  STRUCT
   S700 : STRUCT
    M_AUTO_SEL : BOOL ;
    M_MANUAL_SEL : BOOL ;
    M_READY_PB : BOOL ;
    M_AUTO_RUN_PB : BOOL ;
    M_WORK_COMP_SET_PB : BOOL ;
    M_WORK_COMP_RST_PB : BOOL ;
    M_HOME_POS_PB : BOOL ;
    SPARE8 : BOOL ;
    TL_PIN_SEL : BOOL ;
    LM_PIN_SEL : BOOL ;
    TL_LATCH_SEL : BOOL ;
    LM_LATCH_SEL : BOOL ;
    SPARE13 : BOOL ;
    SPARE14 : BOOL ;
    SPARE15 : BOOL ;
    SPARE16 : BOOL ;
    SPARE17 : BOOL ;
    SPARE18 : BOOL ;
    SPARE19 : BOOL ;
    SPARE20 : BOOL ;
    SPARE21 : BOOL ;
    SPARE22 : BOOL ;
    SPARE23 : BOOL ;
    SPARE24 : BOOL ;
    SPARE25 : BOOL ;
    SPARE26 : BOOL ;
    SPARE27 : BOOL ;
    SPARE28 : BOOL ;
    SPARE29 : BOOL ;
    SPARE30 : BOOL ;
    M_ADV_PB : BOOL ;
    M_RET_PB : BOOL ;
    SPARE34 : BOOL ;
    SPARE35 : BOOL ;
    SPARE36 : BOOL ;
    SPARE37 : BOOL ;
    M_RBT_WORK_COMP_SET_PB : BOOL ;
    M_RBT_WORK_COMP_RST_PB : BOOL ;
    SPARE40 : BOOL ;
    SPARE41 : BOOL ;
    SPARE42 : BOOL ;
    SPARE43 : BOOL ;
    SPARE44 : BOOL ;
    SPARE45 : BOOL ;
    SPARE46 : BOOL ;
    SPARE47 : BOOL ;
    SPARE48 : BOOL ;
    SPARE49 : BOOL ;
    SPARE50 : BOOL ;
    SPARE51 : BOOL ;
    SPARE52 : BOOL ;
    SPARE53 : BOOL ;
    SPARE54 : BOOL ;
    SPARE55 : BOOL ;
    SPARE56 : BOOL ;
    SPARE57 : BOOL ;
    SPARE58 : BOOL ;
    SPARE59 : BOOL ;
    SPARE60 : BOOL ;
    SPARE61 : BOOL ;
    SPARE62 : BOOL ;
    SPARE63 : BOOL ;
    SPARE64 : BOOL ;
    SPARE65 : BOOL ;
    SPARE66 : BOOL ;
    SPARE67 : BOOL ;
    SPARE68 : BOOL ;
    SPARE69 : BOOL ;
    SPARE70 : BOOL ;
    SPARE71 : BOOL ;
    SPARE72 : BOOL ;
    SPARE73 : BOOL ;
    SPARE74 : BOOL ;
    SPARE75 : BOOL ;
    SPARE76 : BOOL ;
    SPARE77 : BOOL ;
    SPARE78 : BOOL ;
    SPARE79 : BOOL ;
    SPARE80 : BOOL ;
    SPARE81 : BOOL ;
    SPARE82 : BOOL ;
    SPARE83 : BOOL ;
    SPARE84 : BOOL ;
    SPARE85 : BOOL ;
    SPARE86 : BOOL ;
    SPARE87 : BOOL ;
    SPARE88 : BOOL ;
    SPARE89 : BOOL ;
    SPARE90 : BOOL ;
    SPARE91 : BOOL ;
    SPARE92 : BOOL ;
    SPARE93 : BOOL ;
    SPARE94 : BOOL ;
    SPARE95 : BOOL ;
    SPARE96 : BOOL ;
    SPARE97 : BOOL ;
    SPARE98 : BOOL ;
    SPARE99 : BOOL ;
    SPARE100 : BOOL ;
    SPARE101 : BOOL ;
    SPARE102 : BOOL ;
    SPARE103 : BOOL ;
    SPARE104 : BOOL ;
    SPARE105 : BOOL ;
    SPARE106 : BOOL ;
    SPARE107 : BOOL ;
    SPARE108 : BOOL ;
    SPARE109 : BOOL ;
    SPARE110 : BOOL ;
    SPARE111 : BOOL ;
    SPARE112 : BOOL ;
    SPARE113 : BOOL ;
    SPARE114 : BOOL ;
    SPARE115 : BOOL ;
    SPARE116 : BOOL ;
    SPARE117 : BOOL ;
    SPARE118 : BOOL ;
    SPARE119 : BOOL ;
    SPARE120 : BOOL ;
    SPARE121 : BOOL ;
    SPARE122 : BOOL ;
    SPARE123 : BOOL ;
    SPARE124 : BOOL ;
    SPARE125 : BOOL ;
    SPARE126 : BOOL ;
    SPARE127 : BOOL ;
    SPARE128 : BOOL ;
    SPARE129 : BOOL ;
    SPARE130 : BOOL ;
    SPARE131 : BOOL ;
    SPARE132 : BOOL ;
    SPARE133 : BOOL ;
    SPARE134 : BOOL ;
    SPARE135 : BOOL ;
    SPARE136 : BOOL ;
    SPARE137 : BOOL ;
    SPARE138 : BOOL ;
    SPARE139 : BOOL ;
    SPARE140 : BOOL ;
    SPARE141 : BOOL ;
    SPARE142 : BOOL ;
    SPARE143 : BOOL ;
    SPARE144 : BOOL ;
    SPARE145 : BOOL ;
    SPARE146 : BOOL ;
    SPARE147 : BOOL ;
    SPARE148 : BOOL ;
    SPARE149 : BOOL ;
    SPARE150 : BOOL ;
    SPARE151 : BOOL ;
    SPARE152 : BOOL ;
    SPARE153 : BOOL ;
    SPARE154 : BOOL ;
    SPARE155 : BOOL ;
    SPARE156 : BOOL ;
    SPARE157 : BOOL ;
    SPARE158 : BOOL ;
    SPARE159 : BOOL ;
    SPARE160 : BOOL ;
    SPARE161 : BOOL ;
    TL_PIN_UP_LAMP : WORD ;
    TL_PIN_DOWN_LAMP : WORD ;
    LM_PIN_UP_LAMP : WORD ;
    LM_PIN_DOWN_LAMP : WORD ;
    TL_LATCH_ADV_LAMP : WORD ;
    TL_LATCH_RET_LAMP : WORD ;
    LM_LATCH_ADV_LAMP : WORD ;
    LM_LATCH_RET_LAMP : WORD ;
    SP_WORD19 : WORD ;
    SP_WORD20 : WORD ;
    SP_WORD21 : WORD ;
    SP_WORD22 : WORD ;
    SP_WORD23 : WORD ;
    SP_WORD24 : WORD ;
    SP_WORD25 : WORD ;
    SP_WORD26 : WORD ;
    SP_WORD27 : WORD ;
    SP_WORD28 : WORD ;
    SP_WORD29 : WORD ;
    SP_WORD30 : WORD ;
    SP_WORD31 : WORD ;
    SP_WORD32 : WORD ;
    SP_WORD33 : WORD ;
    SP_WORD34 : WORD ;
    SP_WORD36 : WORD ;
    SP_WORD37 : WORD ;
    SP_WORD38 : WORD ;
    SP_WORD39 : WORD ;
    SP_WORD40 : WORD ;
    SP_WORD41 : WORD ;
    SP_WORD42 : WORD ;
    SP_WORD43 : WORD ;
    SP_WORD44 : WORD ;
    SP_WORD45 : WORD ;
    SP_WORD46 : WORD ;
    SP_WORD47 : WORD ;
    SP_WORD48 : WORD ;
    SP_WORD49 : WORD ;
    SP_WORD50 : WORD ;
    SP_WORD51 : WORD ;
    SP_WORD52 : WORD ;
    SP_WORD53 : WORD ;
    SP_WORD54 : WORD ;
    SP_WORD55 : WORD ;
    SP_WORD56 : WORD ;
    SP_WORD57 : WORD ;
    SP_WORD58 : WORD ;
    SP_WORD59 : WORD ;
    SP_WORD60 : WORD ;
    SP_WORD61 : WORD ;
    SP_WORD62 : WORD ;
    SP_WORD63 : WORD ;
    SP_WORD64 : WORD ;
    SP_WORD65 : WORD ;
    SP_WORD66 : WORD ;
    SP_WORD67 : WORD ;
    SP_WORD68 : WORD ;
    SP_WORD69 : WORD ;
    SP_WORD70 : WORD ;
    SP_WORD71 : WORD ;
    SP_WORD72 : WORD ;
    SP_WORD73 : WORD ;
    SP_WORD74 : WORD ;
    SP_WORD75 : WORD ;
    SP_WORD76 : WORD ;
    SP_WORD77 : WORD ;
    SP_WORD78 : WORD ;
    SP_WORD79 : WORD ;
    SP_WORD80 : WORD ;
    SP_WORD81 : WORD ;
    SP_WORD82 : WORD ;
    SP_WORD83 : WORD ;
    SP_WORD84 : WORD ;
    SP_WORD85 : WORD ;
    SP_WORD86 : WORD ;
    SP_WORD87 : WORD ;
    SP_WORD88 : WORD ;
    SP_WORD89 : WORD ;
    SP_WORD90 : WORD ;
    SP_WORD91 : WORD ;
    SP_WORD92 : WORD ;
    SP_WORD93 : WORD ;
    SP_WORD94 : WORD ;
    SP_WORD95 : WORD ;
    SP_WORD96 : WORD ;
    SP_WORD97 : WORD ;
    SP_WORD98 : WORD ;
    SP_WORD99 : WORD ;
    SP_WORD100 : WORD ;
    SP_WORD101 : WORD ;
   END_STRUCT ;
   S701 : STRUCT
    M_AUTO_SEL : BOOL ;
    M_MANUAL_SEL : BOOL ;
    M_READY_PB : BOOL ;
    M_AUTO_RUN_PB : BOOL ;
    M_WORK_COMP_SET_PB : BOOL ;
    M_WORK_COMP_RST_PB : BOOL ;
    M_HOME_POS_PB : BOOL ;
    M_TIP_DRESS_PB : BOOL ;
    INDEX_RET_LOCK_SEL : BOOL ;
    INDEX_ADV_RET_SEL : BOOL ;
    INDEX_ADV_LOCK_SEL : BOOL ;
    SPARE12 : BOOL ;
    SPARE13 : BOOL ;
    SPARE14 : BOOL ;
    SPARE15 : BOOL ;
    SPARE16 : BOOL ;
    SPARE17 : BOOL ;
    SPARE18 : BOOL ;
    SPARE19 : BOOL ;
    SPARE20 : BOOL ;
    SPARE21 : BOOL ;
    SPARE22 : BOOL ;
    SPARE23 : BOOL ;
    SPARE24 : BOOL ;
    SPARE25 : BOOL ;
    SPARE26 : BOOL ;
    SPARE27 : BOOL ;
    SPARE28 : BOOL ;
    SPARE29 : BOOL ;
    SPARE30 : BOOL ;
    M_ADV_PB : BOOL ;
    M_RET_PB : BOOL ;
    LM_INDEX_PIN1_SEL : BOOL ;
    LM_INDEX_PIN2_SEL : BOOL ;
    LM_INDEX_PIN3_SEL : BOOL ;
    LM_INDEX_1_CLAMP1_SEL : BOOL ;
    LM_INDEX_1_CLAMP2_SEL : BOOL ;
    LM_INDEX_1_CLAMP3_SEL : BOOL ;
    LM_INDEX_1_CLAMP4_SEL : BOOL ;
    LM_INDEX_2_CLAMP1_SEL : BOOL ;
    LM_INDEX_2_CLAMP2_SEL : BOOL ;
    LM_INDEX_2_CLAMP3_SEL : BOOL ;
    LM_INDEX_2_CLAMP4_SEL : BOOL ;
    LM_INDEX_2_CLAMP5_SEL : BOOL ;
    LM_INDEX_FDR_SHIFT_SEL : BOOL ;
    LM_INDEX_FDR_PIN_SEL : BOOL ;
    LM_INDEX_ADV_PB : BOOL ;
    LM_INDEX_RET_PB : BOOL ;
    TL_INDEX_PIN1_SEL : BOOL ;
    TL_INDEX_PIN2_SEL : BOOL ;
    TL_INDEX_LOCATE1_SEL : BOOL ;
    TL_INDEX_LOCATE2_SEL : BOOL ;
    TL_INDEX_LOCATE3_SEL : BOOL ;
    TL_INDEX_1_CLAMP1_SEL : BOOL ;
    TL_INDEX_1_CLAMP2_SEL : BOOL ;
    TL_INDEX_CLAMP2_SEL : BOOL ;
    TL_INDEX_CLAMP3_SEL : BOOL ;
    TL_INDEX_CLAMP4_SEL : BOOL ;
    TL_INDEX_FDR_SHIFT_SEL : BOOL ;
    SPARE61 : BOOL ;
    SPARE62 : BOOL ;
    SPARE63 : BOOL ;
    TL_INDEX_ADV_PB : BOOL ;
    TL_INDEX_RET_PB : BOOL ;
    SPARE66 : BOOL ;
    SPARE67 : BOOL ;
    SPARE68 : BOOL ;
    SPARE69 : BOOL ;
    SPARE70 : BOOL ;
    SPARE71 : BOOL ;
    SPARE72 : BOOL ;
    SPARE73 : BOOL ;
    SPARE74 : BOOL ;
    SPARE75 : BOOL ;
    SPARE76 : BOOL ;
    SPARE77 : BOOL ;
    SPARE78 : BOOL ;
    SPARE79 : BOOL ;
    SPARE80 : BOOL ;
    SPARE81 : BOOL ;
    SPARE82 : BOOL ;
    SPARE83 : BOOL ;
    SPARE84 : BOOL ;
    SPARE85 : BOOL ;
    SPARE86 : BOOL ;
    SPARE87 : BOOL ;
    SPARE88 : BOOL ;
    SPARE89 : BOOL ;
    SPARE90 : BOOL ;
    SPARE91 : BOOL ;
    SPARE92 : BOOL ;
    SPARE93 : BOOL ;
    SPARE94 : BOOL ;
    SPARE95 : BOOL ;
    SPARE96 : BOOL ;
    SPARE97 : BOOL ;
    SPARE98 : BOOL ;
    SPARE99 : BOOL ;
    SPARE100 : BOOL ;
    SPARE101 : BOOL ;
    SPARE102 : BOOL ;
    SPARE103 : BOOL ;
    SPARE104 : BOOL ;
    SPARE105 : BOOL ;
    SPARE106 : BOOL ;
    SPARE107 : BOOL ;
    SPARE108 : BOOL ;
    SPARE109 : BOOL ;
    SPARE110 : BOOL ;
    SPARE111 : BOOL ;
    SPARE112 : BOOL ;
    SPARE113 : BOOL ;
    SPARE114 : BOOL ;
    SPARE115 : BOOL ;
    SPARE116 : BOOL ;
    SPARE117 : BOOL ;
    SPARE118 : BOOL ;
    SPARE119 : BOOL ;
    SPARE120 : BOOL ;
    SPARE121 : BOOL ;
    SPARE122 : BOOL ;
    SPARE123 : BOOL ;
    SPARE124 : BOOL ;
    SPARE125 : BOOL ;
    SPARE126 : BOOL ;
    SPARE127 : BOOL ;
    SPARE128 : BOOL ;
    SPARE129 : BOOL ;
    SPARE130 : BOOL ;
    SPARE131 : BOOL ;
    SPARE132 : BOOL ;
    SPARE133 : BOOL ;
    SPARE134 : BOOL ;
    SPARE135 : BOOL ;
    SPARE136 : BOOL ;
    SPARE137 : BOOL ;
    SPARE138 : BOOL ;
    SPARE139 : BOOL ;
    SPARE140 : BOOL ;
    SPARE141 : BOOL ;
    SPARE142 : BOOL ;
    SPARE143 : BOOL ;
    SPARE144 : BOOL ;
    SPARE145 : BOOL ;
    SPARE146 : BOOL ;
    SPARE147 : BOOL ;
    SPARE148 : BOOL ;
    SPARE149 : BOOL ;
    SPARE150 : BOOL ;
    SPARE151 : BOOL ;
    SPARE152 : BOOL ;
    SPARE153 : BOOL ;
    SPARE154 : BOOL ;
    SPARE155 : BOOL ;
    SPARE156 : BOOL ;
    SPARE157 : BOOL ;
    SPARE158 : BOOL ;
    SPARE159 : BOOL ;
    SPARE160 : BOOL ;
    SPARE161 : BOOL ;
    RETURN_LOCK_ADV_LP : WORD ;
    RETURN_LOCK_RET_LP : WORD ;
    INDEX_ADV_LP : WORD ;
    INDEX_RET_LP : WORD ;
    TURN_LOCK_ADV_LP : WORD ;
    TURN_LOCK_RET_LP : WORD ;
    SP_WORD17 : WORD ;
    SP_WORD18 : WORD ;
    SP_WORD19 : WORD ;
    SP_WORD20 : WORD ;
    LM_INDEX_PIN1_UP_LP : WORD ;
    LM_INDEX_PIN1_DOWN_LP : WORD ;
    LM_INDEX_PIN2_UP_LP : WORD ;
    LM_INDEX_PIN2_DOWN_LP : WORD ;
    LM_INDEX_PIN3_UP_LP : WORD ;
    LM_INDEX_PIN3_DOWN_LP : WORD ;
    LM_INDEX_1_CLAMP1_ADV_LP : WORD ;
    LM_INDEX_1_CLAMP1_RET_LP : WORD ;
    LM_INDEX_1_CLAMP2_ADV_LP : WORD ;
    LM_INDEX_1_CLAMP2_RET_LP : WORD ;
    LM_INDEX_1_CLAMP3_ADV_LP : WORD ;
    LM_INDEX_1_CLAMP3_RET_LP : WORD ;
    LM_INDEX_1_CLAMP4_ADV_LP : WORD ;
    LM_INDEX_1_CLAMP4_RET_LP : WORD ;
    LM_INDEX_2_CLAMP1_ADV_LP : WORD ;
    LM_INDEX_2_CLAMP1_RET_LP : WORD ;
    LM_INDEX_2_CLAMP2_ADV_LP : WORD ;
    LM_INDEX_2_CLAMP2_RET_LP : WORD ;
    LM_INDEX_2_CLAMP3_ADV_LP : WORD ;
    LM_INDEX_2_CLAMP3_RET_LP : WORD ;
    LM_INDEX_2_CLAMP4_ADV_LP : WORD ;
    LM_INDEX_2_CLAMP4_RET_LP : WORD ;
    LM_INDEX_2_CLAMP5_ADV_LP : WORD ;
    LM_INDEX_2_CLAMP5_RET_LP : WORD ;
    LM_INDEX_FDR_SFT_ADV_LP : WORD ;
    LM_INDEX_FDR_SFT_RET_LP : WORD ;
    LM_INDEX_FDR_PIN_ADV_LP : WORD ;
    LM_INDEX_FDR_PIN_RET_LP : WORD ;
    SP_WORD50 : WORD ;
    SP_WORD51 : WORD ;
    TL_INDEX_PIN1_UP_LP : WORD ;
    TL_INDEX_PIN1_DOWN_LP : WORD ;
    TL_INDEX_PIN2_UP_LP : WORD ;
    TL_INDEX_PIN2_DOWN_LP : WORD ;
    TL_INDEX_LOCATE1_ADV_LP : WORD ;
    TL_INDEX_LOCATE1_RET_LP : WORD ;
    TL_INDEX_LOCATE2_ADV_LP : WORD ;
    TL_INDEX_LOCATE2_RET_LP : WORD ;
    TL_INDEX_LOCATE3_ADV_LP : WORD ;
    TL_INDEX_LOCATE3_RET_LP : WORD ;
    TL_INDEX_1_CLAMP1_ADV_LP : WORD ;
    TL_INDEX_1_CLAMP1_RET_LP : WORD ;
    TL_INDEX_1_CLAMP2_ADV_LP : WORD ;
    TL_INDEX_1_CLAMP2_RET_LP : WORD ;
    TL_INDEX_CLAMP2_ADV_LP : WORD ;
    TL_INDEX_CLAMP2_RET_LP : WORD ;
    TL_INDEX_CLAMP3_ADV_LP : WORD ;
    TL_INDEX_CLAMP3_RET_LP : WORD ;
    TL_INDEX_CLAMP4_ADV_LP : WORD ;
    TL_INDEX_CLAMP4_RET_LP : WORD ;
    TL_INDEX_FDR_SFT_ADV_LP : WORD ;
    TL_INDEX_FDR_SFT_RET_LP : WORD ;
    SP_WORD74 : WORD ;
    SP_WORD75 : WORD ;
    SP_WORD76 : WORD ;
    SP_WORD77 : WORD ;
    SP_WORD78 : WORD ;
    SP_WORD79 : WORD ;
    SP_WORD80 : WORD ;
    SP_WORD81 : WORD ;
    SP_WORD82 : WORD ;
    SP_WORD83 : WORD ;
    SP_WORD84 : WORD ;
    SP_WORD85 : WORD ;
    SP_WORD86 : WORD ;
    SP_WORD87 : WORD ;
    SP_WORD88 : WORD ;
    SP_WORD89 : WORD ;
    SP_WORD90 : WORD ;
    SP_WORD91 : WORD ;
    SP_WORD92 : WORD ;
    SP_WORD93 : WORD ;
    SP_WORD94 : WORD ;
    SP_WORD95 : WORD ;
    SP_WORD96 : WORD ;
    SP_WORD97 : WORD ;
    SP_WORD98 : WORD ;
    SP_WORD99 : WORD ;
    SP_WORD100 : WORD ;
    SP_WORD101 : WORD ;
   END_STRUCT ;
   S_EXTN : STRUCT
    M_AUTO_SEL : BOOL ;
    M_MANUAL_SEL : BOOL ;
    M_READY_PB : BOOL ;
    M_AUTO_RUN_PB : BOOL ;
    M_WORK_COMP_SET_PB : BOOL ;
    M_WORK_COMP_RST_PB : BOOL ;
    M_HOME_POS_PB : BOOL ;
    SPARE8 : BOOL ;
    LM_STORAGE_UP_DN_SEL : BOOL ;
    LM_EJECT_SEL : BOOL ;
    LM_STORAGE_ADV_RET_SEL : BOOL ;
    TL_STORAGE_UP_DN_SEL : BOOL ;
    TL_EJECT_SEL : BOOL ;
    TL_STORAGE_ADV_RET_SEL : BOOL ;
    BRKT_STORAGE_A_SEL : BOOL ;
    BRKT_STORAGE_B_SEL : BOOL ;
    SPARE17 : BOOL ;
    SPARE18 : BOOL ;
    SPARE19 : BOOL ;
    SPARE20 : BOOL ;
    SPARE21 : BOOL ;
    SPARE22 : BOOL ;
    SPARE23 : BOOL ;
    SPARE24 : BOOL ;
    SPARE25 : BOOL ;
    SPARE26 : BOOL ;
    SPARE27 : BOOL ;
    SPARE28 : BOOL ;
    SPARE29 : BOOL ;
    SPARE30 : BOOL ;
    M_ADV_PB : BOOL ;
    M_RET_PB : BOOL ;
    SPARE34 : BOOL ;
    SPARE35 : BOOL ;
    SPARE36 : BOOL ;
    SPARE37 : BOOL ;
    SPARE38 : BOOL ;
    SPARE39 : BOOL ;
    SPARE40 : BOOL ;
    SPARE41 : BOOL ;
    SPARE42 : BOOL ;
    SPARE43 : BOOL ;
    SPARE44 : BOOL ;
    SPARE45 : BOOL ;
    SPARE46 : BOOL ;
    SPARE47 : BOOL ;
    SPARE48 : BOOL ;
    SPARE49 : BOOL ;
    SPARE50 : BOOL ;
    SPARE51 : BOOL ;
    SPARE52 : BOOL ;
    SPARE53 : BOOL ;
    SPARE54 : BOOL ;
    SPARE55 : BOOL ;
    SPARE56 : BOOL ;
    SPARE57 : BOOL ;
    SPARE58 : BOOL ;
    SPARE59 : BOOL ;
    SPARE60 : BOOL ;
    SPARE61 : BOOL ;
    SPARE62 : BOOL ;
    SPARE63 : BOOL ;
    SPARE64 : BOOL ;
    SPARE65 : BOOL ;
    SPARE66 : BOOL ;
    SPARE67 : BOOL ;
    SPARE68 : BOOL ;
    SPARE69 : BOOL ;
    SPARE70 : BOOL ;
    SPARE71 : BOOL ;
    SPARE72 : BOOL ;
    SPARE73 : BOOL ;
    SPARE74 : BOOL ;
    SPARE75 : BOOL ;
    SPARE76 : BOOL ;
    SPARE77 : BOOL ;
    SPARE78 : BOOL ;
    SPARE79 : BOOL ;
    SPARE80 : BOOL ;
    SPARE81 : BOOL ;
    SPARE82 : BOOL ;
    SPARE83 : BOOL ;
    SPARE84 : BOOL ;
    SPARE85 : BOOL ;
    SPARE86 : BOOL ;
    SPARE87 : BOOL ;
    SPARE88 : BOOL ;
    SPARE89 : BOOL ;
    SPARE90 : BOOL ;
    SPARE91 : BOOL ;
    SPARE92 : BOOL ;
    SPARE93 : BOOL ;
    SPARE94 : BOOL ;
    SPARE95 : BOOL ;
    SPARE96 : BOOL ;
    SPARE97 : BOOL ;
    SPARE98 : BOOL ;
    SPARE99 : BOOL ;
    SPARE100 : BOOL ;
    SPARE101 : BOOL ;
    SPARE102 : BOOL ;
    SPARE103 : BOOL ;
    SPARE104 : BOOL ;
    SPARE105 : BOOL ;
    SPARE106 : BOOL ;
    SPARE107 : BOOL ;
    SPARE108 : BOOL ;
    SPARE109 : BOOL ;
    SPARE110 : BOOL ;
    SPARE111 : BOOL ;
    SPARE112 : BOOL ;
    SPARE113 : BOOL ;
    SPARE114 : BOOL ;
    SPARE115 : BOOL ;
    SPARE116 : BOOL ;
    SPARE117 : BOOL ;
    SPARE118 : BOOL ;
    SPARE119 : BOOL ;
    SPARE120 : BOOL ;
    SPARE121 : BOOL ;
    SPARE122 : BOOL ;
    SPARE123 : BOOL ;
    SPARE124 : BOOL ;
    SPARE125 : BOOL ;
    SPARE126 : BOOL ;
    SPARE127 : BOOL ;
    SPARE128 : BOOL ;
    SPARE129 : BOOL ;
    SPARE130 : BOOL ;
    SPARE131 : BOOL ;
    SPARE132 : BOOL ;
    SPARE133 : BOOL ;
    SPARE134 : BOOL ;
    SPARE135 : BOOL ;
    SPARE136 : BOOL ;
    SPARE137 : BOOL ;
    SPARE138 : BOOL ;
    SPARE139 : BOOL ;
    SPARE140 : BOOL ;
    SPARE141 : BOOL ;
    SPARE142 : BOOL ;
    SPARE143 : BOOL ;
    SPARE144 : BOOL ;
    SPARE145 : BOOL ;
    SPARE146 : BOOL ;
    SPARE147 : BOOL ;
    SPARE148 : BOOL ;
    SPARE149 : BOOL ;
    SPARE150 : BOOL ;
    SPARE151 : BOOL ;
    SPARE152 : BOOL ;
    SPARE153 : BOOL ;
    SPARE154 : BOOL ;
    SPARE155 : BOOL ;
    SPARE156 : BOOL ;
    SPARE157 : BOOL ;
    SPARE158 : BOOL ;
    SPARE159 : BOOL ;
    SPARE160 : BOOL ;
    SPARE161 : BOOL ;
    BRKT_STORAGE_A_ADV_LAMP : WORD ;
    BRKT_STORAGE_A_RET_LAMP : WORD ;
    BRKT_STORAGE_B_ADV_LAMP : WORD ;
    BRKT_STORAGE_B_RET_LAMP : WORD ;
    SP_WORD15 : WORD ;
    SP_WORD16 : WORD ;
    SP_WORD17 : WORD ;
    SP_WORD18 : WORD ;
    SP_WORD19 : WORD ;
    SP_WORD20 : WORD ;
    LM_STORAGE_UP_LAMP : WORD ;
    LM_STORAGE_DOWN_LAMP : WORD ;
    LM_EJECT_UP_LAMP : WORD ;
    LM_EJECT_DOWN_LAMP : WORD ;
    LM_STORAGE_ADV_LAMP : WORD ;
    LM_STORAGE_RET_LAMP : WORD ;
    SP_WORD27 : WORD ;
    SP_WORD28 : WORD ;
    SP_WORD29 : WORD ;
    SP_WORD30 : WORD ;
    TL_STORAGE_UP_LAMP : WORD ;
    TL_STORAGE_DOWN_LAMP : WORD ;
    TL_EJECT_UP_LAMP : WORD ;
    TL_EJECT_DOWN_LAMP : WORD ;
    TL_STORAGE_ADV_LAMP : WORD ;
    TL_STORAGE_RET_LAMP : WORD ;
    SP_WORD38 : WORD ;
    SP_WORD39 : WORD ;
    SP_WORD40 : WORD ;
    SP_WORD41 : WORD ;
    SP_WORD42 : WORD ;
    SP_WORD43 : WORD ;
    SP_WORD44 : WORD ;
    SP_WORD45 : WORD ;
    SP_WORD46 : WORD ;
    SP_WORD47 : WORD ;
    SP_WORD48 : WORD ;
    SP_WORD49 : WORD ;
    SP_WORD50 : WORD ;
    SP_WORD51 : WORD ;
    SP_WORD52 : WORD ;
    SP_WORD53 : WORD ;
    SP_WORD54 : WORD ;
    SP_WORD55 : WORD ;
    SP_WORD56 : WORD ;
    SP_WORD57 : WORD ;
    SP_WORD58 : WORD ;
    SP_WORD59 : WORD ;
    SP_WORD60 : WORD ;
    SP_WORD61 : WORD ;
    SP_WORD62 : WORD ;
    SP_WORD63 : WORD ;
    SP_WORD64 : WORD ;
    SP_WORD65 : WORD ;
    SP_WORD66 : WORD ;
    SP_WORD67 : WORD ;
    SP_WORD68 : WORD ;
    SP_WORD69 : WORD ;
    SP_WORD70 : WORD ;
    SP_WORD71 : WORD ;
    SP_WORD72 : WORD ;
    SP_WORD73 : WORD ;
    SP_WORD74 : WORD ;
    SP_WORD75 : WORD ;
    SP_WORD76 : WORD ;
    SP_WORD77 : WORD ;
    SP_WORD78 : WORD ;
    SP_WORD79 : WORD ;
    SP_WORD80 : WORD ;
    SP_WORD81 : WORD ;
    SP_WORD82 : WORD ;
    SP_WORD83 : WORD ;
    SP_WORD84 : WORD ;
    SP_WORD85 : WORD ;
    SP_WORD86 : WORD ;
    SP_WORD87 : WORD ;
    SP_WORD88 : WORD ;
    SP_WORD89 : WORD ;
    SP_WORD90 : WORD ;
    SP_WORD91 : WORD ;
    SP_WORD92 : WORD ;
    SP_WORD93 : WORD ;
    SP_WORD94 : WORD ;
    SP_WORD95 : WORD ;
    SP_WORD96 : WORD ;
    SP_WORD97 : WORD ;
    SP_WORD98 : WORD ;
    SP_WORD99 : WORD ;
    SP_WORD100 : WORD ;
    SP_WORD101 : WORD ;
   END_STRUCT ;
  END_STRUCT ;
BEGIN
   S700.M_AUTO_SEL := FALSE;
   S700.M_MANUAL_SEL := FALSE;
   S700.M_READY_PB := FALSE;
   S700.M_AUTO_RUN_PB := FALSE;
   S700.M_WORK_COMP_SET_PB := FALSE;
   S700.M_WORK_COMP_RST_PB := FALSE;
   S700.M_HOME_POS_PB := FALSE;
   S700.SPARE8 := FALSE;
   S700.TL_PIN_SEL := FALSE;
   S700.LM_PIN_SEL := FALSE;
   S700.TL_LATCH_SEL := FALSE;
   S700.LM_LATCH_SEL := FALSE;
   S700.SPARE13 := FALSE;
   S700.SPARE14 := FALSE;
   S700.SPARE15 := FALSE;
   S700.SPARE16 := FALSE;
   S700.SPARE17 := FALSE;
   S700.SPARE18 := FALSE;
   S700.SPARE19 := FALSE;
   S700.SPARE20 := FALSE;
   S700.SPARE21 := FALSE;
   S700.SPARE22 := FALSE;
   S700.SPARE23 := FALSE;
   S700.SPARE24 := FALSE;
   S700.SPARE25 := FALSE;
   S700.SPARE26 := FALSE;
   S700.SPARE27 := FALSE;
   S700.SPARE28 := FALSE;
   S700.SPARE29 := FALSE;
   S700.SPARE30 := FALSE;
   S700.M_ADV_PB := FALSE;
   S700.M_RET_PB := FALSE;
   S700.SPARE34 := FALSE;
   S700.SPARE35 := FALSE;
   S700.SPARE36 := FALSE;
   S700.SPARE37 := FALSE;
   S700.M_RBT_WORK_COMP_SET_PB := FALSE;
   S700.M_RBT_WORK_COMP_RST_PB := FALSE;
   S700.SPARE40 := FALSE;
   S700.SPARE41 := FALSE;
   S700.SPARE42 := FALSE;
   S700.SPARE43 := FALSE;
   S700.SPARE44 := FALSE;
   S700.SPARE45 := FALSE;
   S700.SPARE46 := FALSE;
   S700.SPARE47 := FALSE;
   S700.SPARE48 := FALSE;
   S700.SPARE49 := FALSE;
   S700.SPARE50 := FALSE;
   S700.SPARE51 := FALSE;
   S700.SPARE52 := FALSE;
   S700.SPARE53 := FALSE;
   S700.SPARE54 := FALSE;
   S700.SPARE55 := FALSE;
   S700.SPARE56 := FALSE;
   S700.SPARE57 := FALSE;
   S700.SPARE58 := FALSE;
   S700.SPARE59 := FALSE;
   S700.SPARE60 := FALSE;
   S700.SPARE61 := FALSE;
   S700.SPARE62 := FALSE;
   S700.SPARE63 := FALSE;
   S700.SPARE64 := FALSE;
   S700.SPARE65 := FALSE;
   S700.SPARE66 := FALSE;
   S700.SPARE67 := FALSE;
   S700.SPARE68 := FALSE;
   S700.SPARE69 := FALSE;
   S700.SPARE70 := FALSE;
   S700.SPARE71 := FALSE;
   S700.SPARE72 := FALSE;
   S700.SPARE73 := FALSE;
   S700.SPARE74 := FALSE;
   S700.SPARE75 := FALSE;
   S700.SPARE76 := FALSE;
   S700.SPARE77 := FALSE;
   S700.SPARE78 := FALSE;
   S700.SPARE79 := FALSE;
   S700.SPARE80 := FALSE;
   S700.SPARE81 := FALSE;
   S700.SPARE82 := FALSE;
   S700.SPARE83 := FALSE;
   S700.SPARE84 := FALSE;
   S700.SPARE85 := FALSE;
   S700.SPARE86 := FALSE;
   S700.SPARE87 := FALSE;
   S700.SPARE88 := FALSE;
   S700.SPARE89 := FALSE;
   S700.SPARE90 := FALSE;
   S700.SPARE91 := FALSE;
   S700.SPARE92 := FALSE;
   S700.SPARE93 := FALSE;
   S700.SPARE94 := FALSE;
   S700.SPARE95 := FALSE;
   S700.SPARE96 := FALSE;
   S700.SPARE97 := FALSE;
   S700.SPARE98 := FALSE;
   S700.SPARE99 := FALSE;
   S700.SPARE100 := FALSE;
   S700.SPARE101 := FALSE;
   S700.SPARE102 := FALSE;
   S700.SPARE103 := FALSE;
   S700.SPARE104 := FALSE;
   S700.SPARE105 := FALSE;
   S700.SPARE106 := FALSE;
   S700.SPARE107 := FALSE;
   S700.SPARE108 := FALSE;
   S700.SPARE109 := FALSE;
   S700.SPARE110 := FALSE;
   S700.SPARE111 := FALSE;
   S700.SPARE112 := FALSE;
   S700.SPARE113 := FALSE;
   S700.SPARE114 := FALSE;
   S700.SPARE115 := FALSE;
   S700.SPARE116 := FALSE;
   S700.SPARE117 := FALSE;
   S700.SPARE118 := FALSE;
   S700.SPARE119 := FALSE;
   S700.SPARE120 := FALSE;
   S700.SPARE121 := FALSE;
   S700.SPARE122 := FALSE;
   S700.SPARE123 := FALSE;
   S700.SPARE124 := FALSE;
   S700.SPARE125 := FALSE;
   S700.SPARE126 := FALSE;
   S700.SPARE127 := FALSE;
   S700.SPARE128 := FALSE;
   S700.SPARE129 := FALSE;
   S700.SPARE130 := FALSE;
   S700.SPARE131 := FALSE;
   S700.SPARE132 := FALSE;
   S700.SPARE133 := FALSE;
   S700.SPARE134 := FALSE;
   S700.SPARE135 := FALSE;
   S700.SPARE136 := FALSE;
   S700.SPARE137 := FALSE;
   S700.SPARE138 := FALSE;
   S700.SPARE139 := FALSE;
   S700.SPARE140 := FALSE;
   S700.SPARE141 := FALSE;
   S700.SPARE142 := FALSE;
   S700.SPARE143 := FALSE;
   S700.SPARE144 := FALSE;
   S700.SPARE145 := FALSE;
   S700.SPARE146 := FALSE;
   S700.SPARE147 := FALSE;
   S700.SPARE148 := FALSE;
   S700.SPARE149 := FALSE;
   S700.SPARE150 := FALSE;
   S700.SPARE151 := FALSE;
   S700.SPARE152 := FALSE;
   S700.SPARE153 := FALSE;
   S700.SPARE154 := FALSE;
   S700.SPARE155 := FALSE;
   S700.SPARE156 := FALSE;
   S700.SPARE157 := FALSE;
   S700.SPARE158 := FALSE;
   S700.SPARE159 := FALSE;
   S700.SPARE160 := FALSE;
   S700.SPARE161 := FALSE;
   S700.TL_PIN_UP_LAMP := W#16#0;
   S700.TL_PIN_DOWN_LAMP := W#16#0;
   S700.LM_PIN_UP_LAMP := W#16#0;
   S700.LM_PIN_DOWN_LAMP := W#16#0;
   S700.TL_LATCH_ADV_LAMP := W#16#0;
   S700.TL_LATCH_RET_LAMP := W#16#0;
   S700.LM_LATCH_ADV_LAMP := W#16#0;
   S700.LM_LATCH_RET_LAMP := W#16#0;
   S700.SP_WORD19 := W#16#0;
   S700.SP_WORD20 := W#16#0;
   S700.SP_WORD21 := W#16#0;
   S700.SP_WORD22 := W#16#0;
   S700.SP_WORD23 := W#16#0;
   S700.SP_WORD24 := W#16#0;
   S700.SP_WORD25 := W#16#0;
   S700.SP_WORD26 := W#16#0;
   S700.SP_WORD27 := W#16#0;
   S700.SP_WORD28 := W#16#0;
   S700.SP_WORD29 := W#16#0;
   S700.SP_WORD30 := W#16#0;
   S700.SP_WORD31 := W#16#0;
   S700.SP_WORD32 := W#16#0;
   S700.SP_WORD33 := W#16#0;
   S700.SP_WORD34 := W#16#0;
   S700.SP_WORD36 := W#16#0;
   S700.SP_WORD37 := W#16#0;
   S700.SP_WORD38 := W#16#0;
   S700.SP_WORD39 := W#16#0;
   S700.SP_WORD40 := W#16#0;
   S700.SP_WORD41 := W#16#0;
   S700.SP_WORD42 := W#16#0;
   S700.SP_WORD43 := W#16#0;
   S700.SP_WORD44 := W#16#0;
   S700.SP_WORD45 := W#16#0;
   S700.SP_WORD46 := W#16#0;
   S700.SP_WORD47 := W#16#0;
   S700.SP_WORD48 := W#16#0;
   S700.SP_WORD49 := W#16#0;
   S700.SP_WORD50 := W#16#0;
   S700.SP_WORD51 := W#16#0;
   S700.SP_WORD52 := W#16#0;
   S700.SP_WORD53 := W#16#0;
   S700.SP_WORD54 := W#16#0;
   S700.SP_WORD55 := W#16#0;
   S700.SP_WORD56 := W#16#0;
   S700.SP_WORD57 := W#16#0;
   S700.SP_WORD58 := W#16#0;
   S700.SP_WORD59 := W#16#0;
   S700.SP_WORD60 := W#16#0;
   S700.SP_WORD61 := W#16#0;
   S700.SP_WORD62 := W#16#0;
   S700.SP_WORD63 := W#16#0;
   S700.SP_WORD64 := W#16#0;
   S700.SP_WORD65 := W#16#0;
   S700.SP_WORD66 := W#16#0;
   S700.SP_WORD67 := W#16#0;
   S700.SP_WORD68 := W#16#0;
   S700.SP_WORD69 := W#16#0;
   S700.SP_WORD70 := W#16#0;
   S700.SP_WORD71 := W#16#0;
   S700.SP_WORD72 := W#16#0;
   S700.SP_WORD73 := W#16#0;
   S700.SP_WORD74 := W#16#0;
   S700.SP_WORD75 := W#16#0;
   S700.SP_WORD76 := W#16#0;
   S700.SP_WORD77 := W#16#0;
   S700.SP_WORD78 := W#16#0;
   S700.SP_WORD79 := W#16#0;
   S700.SP_WORD80 := W#16#0;
   S700.SP_WORD81 := W#16#0;
   S700.SP_WORD82 := W#16#0;
   S700.SP_WORD83 := W#16#0;
   S700.SP_WORD84 := W#16#0;
   S700.SP_WORD85 := W#16#0;
   S700.SP_WORD86 := W#16#0;
   S700.SP_WORD87 := W#16#0;
   S700.SP_WORD88 := W#16#0;
   S700.SP_WORD89 := W#16#0;
   S700.SP_WORD90 := W#16#0;
   S700.SP_WORD91 := W#16#0;
   S700.SP_WORD92 := W#16#0;
   S700.SP_WORD93 := W#16#0;
   S700.SP_WORD94 := W#16#0;
   S700.SP_WORD95 := W#16#0;
   S700.SP_WORD96 := W#16#0;
   S700.SP_WORD97 := W#16#0;
   S700.SP_WORD98 := W#16#0;
   S700.SP_WORD99 := W#16#0;
   S700.SP_WORD100 := W#16#0;
   S700.SP_WORD101 := W#16#0;
   S701.M_AUTO_SEL := FALSE;
   S701.M_MANUAL_SEL := FALSE;
   S701.M_READY_PB := FALSE;
   S701.M_AUTO_RUN_PB := FALSE;
   S701.M_WORK_COMP_SET_PB := FALSE;
   S701.M_WORK_COMP_RST_PB := FALSE;
   S701.M_HOME_POS_PB := FALSE;
   S701.M_TIP_DRESS_PB := FALSE;
   S701.INDEX_RET_LOCK_SEL := FALSE;
   S701.INDEX_ADV_RET_SEL := FALSE;
   S701.INDEX_ADV_LOCK_SEL := FALSE;
   S701.SPARE12 := FALSE;
   S701.SPARE13 := FALSE;
   S701.SPARE14 := FALSE;
   S701.SPARE15 := FALSE;
   S701.SPARE16 := FALSE;
   S701.SPARE17 := FALSE;
   S701.SPARE18 := FALSE;
   S701.SPARE19 := FALSE;
   S701.SPARE20 := FALSE;
   S701.SPARE21 := FALSE;
   S701.SPARE22 := FALSE;
   S701.SPARE23 := FALSE;
   S701.SPARE24 := FALSE;
   S701.SPARE25 := FALSE;
   S701.SPARE26 := FALSE;
   S701.SPARE27 := FALSE;
   S701.SPARE28 := FALSE;
   S701.SPARE29 := FALSE;
   S701.SPARE30 := FALSE;
   S701.M_ADV_PB := FALSE;
   S701.M_RET_PB := FALSE;
   S701.LM_INDEX_PIN1_SEL := FALSE;
   S701.LM_INDEX_PIN2_SEL := FALSE;
   S701.LM_INDEX_PIN3_SEL := FALSE;
   S701.LM_INDEX_1_CLAMP1_SEL := FALSE;
   S701.LM_INDEX_1_CLAMP2_SEL := FALSE;
   S701.LM_INDEX_1_CLAMP3_SEL := FALSE;
   S701.LM_INDEX_1_CLAMP4_SEL := FALSE;
   S701.LM_INDEX_2_CLAMP1_SEL := FALSE;
   S701.LM_INDEX_2_CLAMP2_SEL := FALSE;
   S701.LM_INDEX_2_CLAMP3_SEL := FALSE;
   S701.LM_INDEX_2_CLAMP4_SEL := FALSE;
   S701.LM_INDEX_2_CLAMP5_SEL := FALSE;
   S701.LM_INDEX_FDR_SHIFT_SEL := FALSE;
   S701.LM_INDEX_FDR_PIN_SEL := FALSE;
   S701.LM_INDEX_ADV_PB := FALSE;
   S701.LM_INDEX_RET_PB := FALSE;
   S701.TL_INDEX_PIN1_SEL := FALSE;
   S701.TL_INDEX_PIN2_SEL := FALSE;
   S701.TL_INDEX_LOCATE1_SEL := FALSE;
   S701.TL_INDEX_LOCATE2_SEL := FALSE;
   S701.TL_INDEX_LOCATE3_SEL := FALSE;
   S701.TL_INDEX_1_CLAMP1_SEL := FALSE;
   S701.TL_INDEX_1_CLAMP2_SEL := FALSE;
   S701.TL_INDEX_CLAMP2_SEL := FALSE;
   S701.TL_INDEX_CLAMP3_SEL := FALSE;
   S701.TL_INDEX_CLAMP4_SEL := FALSE;
   S701.TL_INDEX_FDR_SHIFT_SEL := FALSE;
   S701.SPARE61 := FALSE;
   S701.SPARE62 := FALSE;
   S701.SPARE63 := FALSE;
   S701.TL_INDEX_ADV_PB := FALSE;
   S701.TL_INDEX_RET_PB := FALSE;
   S701.SPARE66 := FALSE;
   S701.SPARE67 := FALSE;
   S701.SPARE68 := FALSE;
   S701.SPARE69 := FALSE;
   S701.SPARE70 := FALSE;
   S701.SPARE71 := FALSE;
   S701.SPARE72 := FALSE;
   S701.SPARE73 := FALSE;
   S701.SPARE74 := FALSE;
   S701.SPARE75 := FALSE;
   S701.SPARE76 := FALSE;
   S701.SPARE77 := FALSE;
   S701.SPARE78 := FALSE;
   S701.SPARE79 := FALSE;
   S701.SPARE80 := FALSE;
   S701.SPARE81 := FALSE;
   S701.SPARE82 := FALSE;
   S701.SPARE83 := FALSE;
   S701.SPARE84 := FALSE;
   S701.SPARE85 := FALSE;
   S701.SPARE86 := FALSE;
   S701.SPARE87 := FALSE;
   S701.SPARE88 := FALSE;
   S701.SPARE89 := FALSE;
   S701.SPARE90 := FALSE;
   S701.SPARE91 := FALSE;
   S701.SPARE92 := FALSE;
   S701.SPARE93 := FALSE;
   S701.SPARE94 := FALSE;
   S701.SPARE95 := FALSE;
   S701.SPARE96 := FALSE;
   S701.SPARE97 := FALSE;
   S701.SPARE98 := FALSE;
   S701.SPARE99 := FALSE;
   S701.SPARE100 := FALSE;
   S701.SPARE101 := FALSE;
   S701.SPARE102 := FALSE;
   S701.SPARE103 := FALSE;
   S701.SPARE104 := FALSE;
   S701.SPARE105 := FALSE;
   S701.SPARE106 := FALSE;
   S701.SPARE107 := FALSE;
   S701.SPARE108 := FALSE;
   S701.SPARE109 := FALSE;
   S701.SPARE110 := FALSE;
   S701.SPARE111 := FALSE;
   S701.SPARE112 := FALSE;
   S701.SPARE113 := FALSE;
   S701.SPARE114 := FALSE;
   S701.SPARE115 := FALSE;
   S701.SPARE116 := FALSE;
   S701.SPARE117 := FALSE;
   S701.SPARE118 := FALSE;
   S701.SPARE119 := FALSE;
   S701.SPARE120 := FALSE;
   S701.SPARE121 := FALSE;
   S701.SPARE122 := FALSE;
   S701.SPARE123 := FALSE;
   S701.SPARE124 := FALSE;
   S701.SPARE125 := FALSE;
   S701.SPARE126 := FALSE;
   S701.SPARE127 := FALSE;
   S701.SPARE128 := FALSE;
   S701.SPARE129 := FALSE;
   S701.SPARE130 := FALSE;
   S701.SPARE131 := FALSE;
   S701.SPARE132 := FALSE;
   S701.SPARE133 := FALSE;
   S701.SPARE134 := FALSE;
   S701.SPARE135 := FALSE;
   S701.SPARE136 := FALSE;
   S701.SPARE137 := FALSE;
   S701.SPARE138 := FALSE;
   S701.SPARE139 := FALSE;
   S701.SPARE140 := FALSE;
   S701.SPARE141 := FALSE;
   S701.SPARE142 := FALSE;
   S701.SPARE143 := FALSE;
   S701.SPARE144 := FALSE;
   S701.SPARE145 := FALSE;
   S701.SPARE146 := FALSE;
   S701.SPARE147 := FALSE;
   S701.SPARE148 := FALSE;
   S701.SPARE149 := FALSE;
   S701.SPARE150 := FALSE;
   S701.SPARE151 := FALSE;
   S701.SPARE152 := FALSE;
   S701.SPARE153 := FALSE;
   S701.SPARE154 := FALSE;
   S701.SPARE155 := FALSE;
   S701.SPARE156 := FALSE;
   S701.SPARE157 := FALSE;
   S701.SPARE158 := FALSE;
   S701.SPARE159 := FALSE;
   S701.SPARE160 := FALSE;
   S701.SPARE161 := FALSE;
   S701.RETURN_LOCK_ADV_LP := W#16#0;
   S701.RETURN_LOCK_RET_LP := W#16#0;
   S701.INDEX_ADV_LP := W#16#0;
   S701.INDEX_RET_LP := W#16#0;
   S701.TURN_LOCK_ADV_LP := W#16#0;
   S701.TURN_LOCK_RET_LP := W#16#0;
   S701.SP_WORD17 := W#16#0;
   S701.SP_WORD18 := W#16#0;
   S701.SP_WORD19 := W#16#0;
   S701.SP_WORD20 := W#16#0;
   S701.LM_INDEX_PIN1_UP_LP := W#16#0;
   S701.LM_INDEX_PIN1_DOWN_LP := W#16#0;
   S701.LM_INDEX_PIN2_UP_LP := W#16#0;
   S701.LM_INDEX_PIN2_DOWN_LP := W#16#0;
   S701.LM_INDEX_PIN3_UP_LP := W#16#0;
   S701.LM_INDEX_PIN3_DOWN_LP := W#16#0;
   S701.LM_INDEX_1_CLAMP1_ADV_LP := W#16#0;
   S701.LM_INDEX_1_CLAMP1_RET_LP := W#16#0;
   S701.LM_INDEX_1_CLAMP2_ADV_LP := W#16#0;
   S701.LM_INDEX_1_CLAMP2_RET_LP := W#16#0;
   S701.LM_INDEX_1_CLAMP3_ADV_LP := W#16#0;
   S701.LM_INDEX_1_CLAMP3_RET_LP := W#16#0;
   S701.LM_INDEX_1_CLAMP4_ADV_LP := W#16#0;
   S701.LM_INDEX_1_CLAMP4_RET_LP := W#16#0;
   S701.LM_INDEX_2_CLAMP1_ADV_LP := W#16#0;
   S701.LM_INDEX_2_CLAMP1_RET_LP := W#16#0;
   S701.LM_INDEX_2_CLAMP2_ADV_LP := W#16#0;
   S701.LM_INDEX_2_CLAMP2_RET_LP := W#16#0;
   S701.LM_INDEX_2_CLAMP3_ADV_LP := W#16#0;
   S701.LM_INDEX_2_CLAMP3_RET_LP := W#16#0;
   S701.LM_INDEX_2_CLAMP4_ADV_LP := W#16#0;
   S701.LM_INDEX_2_CLAMP4_RET_LP := W#16#0;
   S701.LM_INDEX_2_CLAMP5_ADV_LP := W#16#0;
   S701.LM_INDEX_2_CLAMP5_RET_LP := W#16#0;
   S701.LM_INDEX_FDR_SFT_ADV_LP := W#16#0;
   S701.LM_INDEX_FDR_SFT_RET_LP := W#16#0;
   S701.LM_INDEX_FDR_PIN_ADV_LP := W#16#0;
   S701.LM_INDEX_FDR_PIN_RET_LP := W#16#0;
   S701.SP_WORD50 := W#16#0;
   S701.SP_WORD51 := W#16#0;
   S701.TL_INDEX_PIN1_UP_LP := W#16#0;
   S701.TL_INDEX_PIN1_DOWN_LP := W#16#0;
   S701.TL_INDEX_PIN2_UP_LP := W#16#0;
   S701.TL_INDEX_PIN2_DOWN_LP := W#16#0;
   S701.TL_INDEX_LOCATE1_ADV_LP := W#16#0;
   S701.TL_INDEX_LOCATE1_RET_LP := W#16#0;
   S701.TL_INDEX_LOCATE2_ADV_LP := W#16#0;
   S701.TL_INDEX_LOCATE2_RET_LP := W#16#0;
   S701.TL_INDEX_LOCATE3_ADV_LP := W#16#0;
   S701.TL_INDEX_LOCATE3_RET_LP := W#16#0;
   S701.TL_INDEX_1_CLAMP1_ADV_LP := W#16#0;
   S701.TL_INDEX_1_CLAMP1_RET_LP := W#16#0;
   S701.TL_INDEX_1_CLAMP2_ADV_LP := W#16#0;
   S701.TL_INDEX_1_CLAMP2_RET_LP := W#16#0;
   S701.TL_INDEX_CLAMP2_ADV_LP := W#16#0;
   S701.TL_INDEX_CLAMP2_RET_LP := W#16#0;
   S701.TL_INDEX_CLAMP3_ADV_LP := W#16#0;
   S701.TL_INDEX_CLAMP3_RET_LP := W#16#0;
   S701.TL_INDEX_CLAMP4_ADV_LP := W#16#0;
   S701.TL_INDEX_CLAMP4_RET_LP := W#16#0;
   S701.TL_INDEX_FDR_SFT_ADV_LP := W#16#0;
   S701.TL_INDEX_FDR_SFT_RET_LP := W#16#0;
   S701.SP_WORD74 := W#16#0;
   S701.SP_WORD75 := W#16#0;
   S701.SP_WORD76 := W#16#0;
   S701.SP_WORD77 := W#16#0;
   S701.SP_WORD78 := W#16#0;
   S701.SP_WORD79 := W#16#0;
   S701.SP_WORD80 := W#16#0;
   S701.SP_WORD81 := W#16#0;
   S701.SP_WORD82 := W#16#0;
   S701.SP_WORD83 := W#16#0;
   S701.SP_WORD84 := W#16#0;
   S701.SP_WORD85 := W#16#0;
   S701.SP_WORD86 := W#16#0;
   S701.SP_WORD87 := W#16#0;
   S701.SP_WORD88 := W#16#0;
   S701.SP_WORD89 := W#16#0;
   S701.SP_WORD90 := W#16#0;
   S701.SP_WORD91 := W#16#0;
   S701.SP_WORD92 := W#16#0;
   S701.SP_WORD93 := W#16#0;
   S701.SP_WORD94 := W#16#0;
   S701.SP_WORD95 := W#16#0;
   S701.SP_WORD96 := W#16#0;
   S701.SP_WORD97 := W#16#0;
   S701.SP_WORD98 := W#16#0;
   S701.SP_WORD99 := W#16#0;
   S701.SP_WORD100 := W#16#0;
   S701.SP_WORD101 := W#16#0;
   S_EXTN.M_AUTO_SEL := FALSE;
   S_EXTN.M_MANUAL_SEL := FALSE;
   S_EXTN.M_READY_PB := FALSE;
   S_EXTN.M_AUTO_RUN_PB := FALSE;
   S_EXTN.M_WORK_COMP_SET_PB := FALSE;
   S_EXTN.M_WORK_COMP_RST_PB := FALSE;
   S_EXTN.M_HOME_POS_PB := FALSE;
   S_EXTN.SPARE8 := FALSE;
   S_EXTN.LM_STORAGE_UP_DN_SEL := FALSE;
   S_EXTN.LM_EJECT_SEL := FALSE;
   S_EXTN.LM_STORAGE_ADV_RET_SEL := FALSE;
   S_EXTN.TL_STORAGE_UP_DN_SEL := FALSE;
   S_EXTN.TL_EJECT_SEL := FALSE;
   S_EXTN.TL_STORAGE_ADV_RET_SEL := FALSE;
   S_EXTN.BRKT_STORAGE_A_SEL := FALSE;
   S_EXTN.BRKT_STORAGE_B_SEL := FALSE;
   S_EXTN.SPARE17 := FALSE;
   S_EXTN.SPARE18 := FALSE;
   S_EXTN.SPARE19 := FALSE;
   S_EXTN.SPARE20 := FALSE;
   S_EXTN.SPARE21 := FALSE;
   S_EXTN.SPARE22 := FALSE;
   S_EXTN.SPARE23 := FALSE;
   S_EXTN.SPARE24 := FALSE;
   S_EXTN.SPARE25 := FALSE;
   S_EXTN.SPARE26 := FALSE;
   S_EXTN.SPARE27 := FALSE;
   S_EXTN.SPARE28 := FALSE;
   S_EXTN.SPARE29 := FALSE;
   S_EXTN.SPARE30 := FALSE;
   S_EXTN.M_ADV_PB := FALSE;
   S_EXTN.M_RET_PB := FALSE;
   S_EXTN.SPARE34 := FALSE;
   S_EXTN.SPARE35 := FALSE;
   S_EXTN.SPARE36 := FALSE;
   S_EXTN.SPARE37 := FALSE;
   S_EXTN.SPARE38 := FALSE;
   S_EXTN.SPARE39 := FALSE;
   S_EXTN.SPARE40 := FALSE;
   S_EXTN.SPARE41 := FALSE;
   S_EXTN.SPARE42 := FALSE;
   S_EXTN.SPARE43 := FALSE;
   S_EXTN.SPARE44 := FALSE;
   S_EXTN.SPARE45 := FALSE;
   S_EXTN.SPARE46 := FALSE;
   S_EXTN.SPARE47 := FALSE;
   S_EXTN.SPARE48 := FALSE;
   S_EXTN.SPARE49 := FALSE;
   S_EXTN.SPARE50 := FALSE;
   S_EXTN.SPARE51 := FALSE;
   S_EXTN.SPARE52 := FALSE;
   S_EXTN.SPARE53 := FALSE;
   S_EXTN.SPARE54 := FALSE;
   S_EXTN.SPARE55 := FALSE;
   S_EXTN.SPARE56 := FALSE;
   S_EXTN.SPARE57 := FALSE;
   S_EXTN.SPARE58 := FALSE;
   S_EXTN.SPARE59 := FALSE;
   S_EXTN.SPARE60 := FALSE;
   S_EXTN.SPARE61 := FALSE;
   S_EXTN.SPARE62 := FALSE;
   S_EXTN.SPARE63 := FALSE;
   S_EXTN.SPARE64 := FALSE;
   S_EXTN.SPARE65 := FALSE;
   S_EXTN.SPARE66 := FALSE;
   S_EXTN.SPARE67 := FALSE;
   S_EXTN.SPARE68 := FALSE;
   S_EXTN.SPARE69 := FALSE;
   S_EXTN.SPARE70 := FALSE;
   S_EXTN.SPARE71 := FALSE;
   S_EXTN.SPARE72 := FALSE;
   S_EXTN.SPARE73 := FALSE;
   S_EXTN.SPARE74 := FALSE;
   S_EXTN.SPARE75 := FALSE;
   S_EXTN.SPARE76 := FALSE;
   S_EXTN.SPARE77 := FALSE;
   S_EXTN.SPARE78 := FALSE;
   S_EXTN.SPARE79 := FALSE;
   S_EXTN.SPARE80 := FALSE;
   S_EXTN.SPARE81 := FALSE;
   S_EXTN.SPARE82 := FALSE;
   S_EXTN.SPARE83 := FALSE;
   S_EXTN.SPARE84 := FALSE;
   S_EXTN.SPARE85 := FALSE;
   S_EXTN.SPARE86 := FALSE;
   S_EXTN.SPARE87 := FALSE;
   S_EXTN.SPARE88 := FALSE;
   S_EXTN.SPARE89 := FALSE;
   S_EXTN.SPARE90 := FALSE;
   S_EXTN.SPARE91 := FALSE;
   S_EXTN.SPARE92 := FALSE;
   S_EXTN.SPARE93 := FALSE;
   S_EXTN.SPARE94 := FALSE;
   S_EXTN.SPARE95 := FALSE;
   S_EXTN.SPARE96 := FALSE;
   S_EXTN.SPARE97 := FALSE;
   S_EXTN.SPARE98 := FALSE;
   S_EXTN.SPARE99 := FALSE;
   S_EXTN.SPARE100 := FALSE;
   S_EXTN.SPARE101 := FALSE;
   S_EXTN.SPARE102 := FALSE;
   S_EXTN.SPARE103 := FALSE;
   S_EXTN.SPARE104 := FALSE;
   S_EXTN.SPARE105 := FALSE;
   S_EXTN.SPARE106 := FALSE;
   S_EXTN.SPARE107 := FALSE;
   S_EXTN.SPARE108 := FALSE;
   S_EXTN.SPARE109 := FALSE;
   S_EXTN.SPARE110 := FALSE;
   S_EXTN.SPARE111 := FALSE;
   S_EXTN.SPARE112 := FALSE;
   S_EXTN.SPARE113 := FALSE;
   S_EXTN.SPARE114 := FALSE;
   S_EXTN.SPARE115 := FALSE;
   S_EXTN.SPARE116 := FALSE;
   S_EXTN.SPARE117 := FALSE;
   S_EXTN.SPARE118 := FALSE;
   S_EXTN.SPARE119 := FALSE;
   S_EXTN.SPARE120 := FALSE;
   S_EXTN.SPARE121 := FALSE;
   S_EXTN.SPARE122 := FALSE;
   S_EXTN.SPARE123 := FALSE;
   S_EXTN.SPARE124 := FALSE;
   S_EXTN.SPARE125 := FALSE;
   S_EXTN.SPARE126 := FALSE;
   S_EXTN.SPARE127 := FALSE;
   S_EXTN.SPARE128 := FALSE;
   S_EXTN.SPARE129 := FALSE;
   S_EXTN.SPARE130 := FALSE;
   S_EXTN.SPARE131 := FALSE;
   S_EXTN.SPARE132 := FALSE;
   S_EXTN.SPARE133 := FALSE;
   S_EXTN.SPARE134 := FALSE;
   S_EXTN.SPARE135 := FALSE;
   S_EXTN.SPARE136 := FALSE;
   S_EXTN.SPARE137 := FALSE;
   S_EXTN.SPARE138 := FALSE;
   S_EXTN.SPARE139 := FALSE;
   S_EXTN.SPARE140 := FALSE;
   S_EXTN.SPARE141 := FALSE;
   S_EXTN.SPARE142 := FALSE;
   S_EXTN.SPARE143 := FALSE;
   S_EXTN.SPARE144 := FALSE;
   S_EXTN.SPARE145 := FALSE;
   S_EXTN.SPARE146 := FALSE;
   S_EXTN.SPARE147 := FALSE;
   S_EXTN.SPARE148 := FALSE;
   S_EXTN.SPARE149 := FALSE;
   S_EXTN.SPARE150 := FALSE;
   S_EXTN.SPARE151 := FALSE;
   S_EXTN.SPARE152 := FALSE;
   S_EXTN.SPARE153 := FALSE;
   S_EXTN.SPARE154 := FALSE;
   S_EXTN.SPARE155 := FALSE;
   S_EXTN.SPARE156 := FALSE;
   S_EXTN.SPARE157 := FALSE;
   S_EXTN.SPARE158 := FALSE;
   S_EXTN.SPARE159 := FALSE;
   S_EXTN.SPARE160 := FALSE;
   S_EXTN.SPARE161 := FALSE;
   S_EXTN.BRKT_STORAGE_A_ADV_LAMP := W#16#0;
   S_EXTN.BRKT_STORAGE_A_RET_LAMP := W#16#0;
   S_EXTN.BRKT_STORAGE_B_ADV_LAMP := W#16#0;
   S_EXTN.BRKT_STORAGE_B_RET_LAMP := W#16#0;
   S_EXTN.SP_WORD15 := W#16#0;
   S_EXTN.SP_WORD16 := W#16#0;
   S_EXTN.SP_WORD17 := W#16#0;
   S_EXTN.SP_WORD18 := W#16#0;
   S_EXTN.SP_WORD19 := W#16#0;
   S_EXTN.SP_WORD20 := W#16#0;
   S_EXTN.LM_STORAGE_UP_LAMP := W#16#0;
   S_EXTN.LM_STORAGE_DOWN_LAMP := W#16#0;
   S_EXTN.LM_EJECT_UP_LAMP := W#16#0;
   S_EXTN.LM_EJECT_DOWN_LAMP := W#16#0;
   S_EXTN.LM_STORAGE_ADV_LAMP := W#16#0;
   S_EXTN.LM_STORAGE_RET_LAMP := W#16#0;
   S_EXTN.SP_WORD27 := W#16#0;
   S_EXTN.SP_WORD28 := W#16#0;
   S_EXTN.SP_WORD29 := W#16#0;
   S_EXTN.SP_WORD30 := W#16#0;
   S_EXTN.TL_STORAGE_UP_LAMP := W#16#0;
   S_EXTN.TL_STORAGE_DOWN_LAMP := W#16#0;
   S_EXTN.TL_EJECT_UP_LAMP := W#16#0;
   S_EXTN.TL_EJECT_DOWN_LAMP := W#16#0;
   S_EXTN.TL_STORAGE_ADV_LAMP := W#16#0;
   S_EXTN.TL_STORAGE_RET_LAMP := W#16#0;
   S_EXTN.SP_WORD38 := W#16#0;
   S_EXTN.SP_WORD39 := W#16#0;
   S_EXTN.SP_WORD40 := W#16#0;
   S_EXTN.SP_WORD41 := W#16#0;
   S_EXTN.SP_WORD42 := W#16#0;
   S_EXTN.SP_WORD43 := W#16#0;
   S_EXTN.SP_WORD44 := W#16#0;
   S_EXTN.SP_WORD45 := W#16#0;
   S_EXTN.SP_WORD46 := W#16#0;
   S_EXTN.SP_WORD47 := W#16#0;
   S_EXTN.SP_WORD48 := W#16#0;
   S_EXTN.SP_WORD49 := W#16#0;
   S_EXTN.SP_WORD50 := W#16#0;
   S_EXTN.SP_WORD51 := W#16#0;
   S_EXTN.SP_WORD52 := W#16#0;
   S_EXTN.SP_WORD53 := W#16#0;
   S_EXTN.SP_WORD54 := W#16#0;
   S_EXTN.SP_WORD55 := W#16#0;
   S_EXTN.SP_WORD56 := W#16#0;
   S_EXTN.SP_WORD57 := W#16#0;
   S_EXTN.SP_WORD58 := W#16#0;
   S_EXTN.SP_WORD59 := W#16#0;
   S_EXTN.SP_WORD60 := W#16#0;
   S_EXTN.SP_WORD61 := W#16#0;
   S_EXTN.SP_WORD62 := W#16#0;
   S_EXTN.SP_WORD63 := W#16#0;
   S_EXTN.SP_WORD64 := W#16#0;
   S_EXTN.SP_WORD65 := W#16#0;
   S_EXTN.SP_WORD66 := W#16#0;
   S_EXTN.SP_WORD67 := W#16#0;
   S_EXTN.SP_WORD68 := W#16#0;
   S_EXTN.SP_WORD69 := W#16#0;
   S_EXTN.SP_WORD70 := W#16#0;
   S_EXTN.SP_WORD71 := W#16#0;
   S_EXTN.SP_WORD72 := W#16#0;
   S_EXTN.SP_WORD73 := W#16#0;
   S_EXTN.SP_WORD74 := W#16#0;
   S_EXTN.SP_WORD75 := W#16#0;
   S_EXTN.SP_WORD76 := W#16#0;
   S_EXTN.SP_WORD77 := W#16#0;
   S_EXTN.SP_WORD78 := W#16#0;
   S_EXTN.SP_WORD79 := W#16#0;
   S_EXTN.SP_WORD80 := W#16#0;
   S_EXTN.SP_WORD81 := W#16#0;
   S_EXTN.SP_WORD82 := W#16#0;
   S_EXTN.SP_WORD83 := W#16#0;
   S_EXTN.SP_WORD84 := W#16#0;
   S_EXTN.SP_WORD85 := W#16#0;
   S_EXTN.SP_WORD86 := W#16#0;
   S_EXTN.SP_WORD87 := W#16#0;
   S_EXTN.SP_WORD88 := W#16#0;
   S_EXTN.SP_WORD89 := W#16#0;
   S_EXTN.SP_WORD90 := W#16#0;
   S_EXTN.SP_WORD91 := W#16#0;
   S_EXTN.SP_WORD92 := W#16#0;
   S_EXTN.SP_WORD93 := W#16#0;
   S_EXTN.SP_WORD94 := W#16#0;
   S_EXTN.SP_WORD95 := W#16#0;
   S_EXTN.SP_WORD96 := W#16#0;
   S_EXTN.SP_WORD97 := W#16#0;
   S_EXTN.SP_WORD98 := W#16#0;
   S_EXTN.SP_WORD99 := W#16#0;
   S_EXTN.SP_WORD100 := W#16#0;
   S_EXTN.SP_WORD101 := W#16#0;
END_DATA_BLOCK

DATA_BLOCK DB 52
TITLE =
VERSION : 0.1


  STRUCT
   S700_R1 : STRUCT 	//Temporary placeholder variable
    PREVIOUS_TIME : INT ;
    CURRENT_TIME : INT ;
   END_STRUCT ;
   S700_IDLE : STRUCT 	//Temporary placeholder variable
    PREVIOUS_TIME : INT ;
    CURRENT_TIME : INT ;
   END_STRUCT ;
   S700_R2 : STRUCT 	//Temporary placeholder variable
    PREVIOUS_TIME : INT ;
    CURRENT_TIME : INT ;
   END_STRUCT ;
   S700_1_IDLE : STRUCT 	//Temporary placeholder variable
    PREVIOUS_TIME : INT ;
    CURRENT_TIME : INT ;
   END_STRUCT ;
   S701_R3 : STRUCT 	//Temporary placeholder variable
    PREVIOUS_TIME : INT ;
    CURRENT_TIME : INT ;
   END_STRUCT ;
   S701 : STRUCT 	//Temporary placeholder variable
    PREVIOUS_TIME : INT ;
    CURRENT_TIME : INT ;
   END_STRUCT ;
   S701_R4 : STRUCT 	//Temporary placeholder variable
    PREVIOUS_TIME : INT ;
    CURRENT_TIME : INT ;
   END_STRUCT ;
   SPARE1 : STRUCT 	//Temporary placeholder variable
    PREVIOUS_TIME : INT ;
    CURRENT_TIME : INT ;
   END_STRUCT ;
   SPARE2 : STRUCT 	//Temporary placeholder variable
    PREVIOUS_TIME : INT ;
    CURRENT_TIME : INT ;
   END_STRUCT ;
   SPARE3 : STRUCT 	//Temporary placeholder variable
    PREVIOUS_TIME : INT ;
    CURRENT_TIME : INT ;
   END_STRUCT ;
   SPARE4 : STRUCT 	//Temporary placeholder variable
    PREVIOUS_TIME : INT ;
    CURRENT_TIME : INT ;
   END_STRUCT ;
   SPARE5 : STRUCT 	//Temporary placeholder variable
    PREVIOUS_TIME : INT ;
    CURRENT_TIME : INT ;
   END_STRUCT ;
   SPARE6 : STRUCT 	//Temporary placeholder variable
    PREVIOUS_TIME : INT ;
    CURRENT_TIME : INT ;
   END_STRUCT ;
   SPARE7 : STRUCT 	//Temporary placeholder variable
    PREVIOUS_TIME : INT ;
    CURRENT_TIME : INT ;
   END_STRUCT ;
   SPARE8 : STRUCT 	//Temporary placeholder variable
    PREVIOUS_TIME : INT ;
    CURRENT_TIME : INT ;
   END_STRUCT ;
   SPARE9 : STRUCT 	//Temporary placeholder variable
    PREVIOUS_TIME : INT ;
    CURRENT_TIME : INT ;
   END_STRUCT ;
   SPARE10 : STRUCT 	//Temporary placeholder variable
    PREVIOUS_TIME : INT ;
    CURRENT_TIME : INT ;
   END_STRUCT ;
   SPARE11 : STRUCT 	//Temporary placeholder variable
    PREVIOUS_TIME : INT ;
    CURRENT_TIME : INT ;
   END_STRUCT ;
   SPARE12 : STRUCT 	//Temporary placeholder variable
    PREVIOUS_TIME : INT ;
    CURRENT_TIME : INT ;
   END_STRUCT ;
   SPARE13 : STRUCT 	//Temporary placeholder variable
    PREVIOUS_TIME : INT ;
    CURRENT_TIME : INT ;
   END_STRUCT ;
   SPARE30 : STRUCT 	//Temporary placeholder variable
    PREVIOUS_TIME : INT ;
    CURRENT_TIME : INT ;
   END_STRUCT ;
   SPARE31 : STRUCT 	//Temporary placeholder variable
    COUNT : INT ;
   END_STRUCT ;
   SPARE32 : STRUCT 	//Temporary placeholder variable
    COUNT : INT ;
   END_STRUCT ;
   SPARE14 : STRUCT 	//Temporary placeholder variable
    PREVIOUS_TIME : INT ;
    CURRENT_TIME : INT ;
   END_STRUCT ;
   SPARE15 : STRUCT 	//Temporary placeholder variable
    PREVIOUS_TIME : INT ;
    CURRENT_TIME : INT ;
   END_STRUCT ;
   SPARE16 : STRUCT 	//Temporary placeholder variable
    PREVIOUS_TIME : INT ;
    CURRENT_TIME : INT ;
   END_STRUCT ;
   OUT_TRV : STRUCT 	//Temporary placeholder variable
    PREVIOUS_TIME : INT ;
    CURRENT_TIME : INT ;
   END_STRUCT ;
   S702 : STRUCT 	//Temporary placeholder variable
    PREVIOUS_TIME : INT ;
    CURRENT_TIME : INT ;
   END_STRUCT ;
   S703 : STRUCT 	//Temporary placeholder variable
    PREVIOUS_TIME : INT ;
    CURRENT_TIME : INT ;
   END_STRUCT ;
   S704 : STRUCT 	//Temporary placeholder variable
    PREVIOUS_TIME : INT ;
    CURRENT_TIME : INT ;
   END_STRUCT ;
   S705 : STRUCT 	//Temporary placeholder variable
    PREVIOUS_TIME : INT ;
    CURRENT_TIME : INT ;
   END_STRUCT ;
   S706 : STRUCT 	//Temporary placeholder variable
    PREVIOUS_TIME : INT ;
    CURRENT_TIME : INT ;
   END_STRUCT ;
   S707 : STRUCT 	//Temporary placeholder variable
    PREVIOUS_TIME : INT ;
    CURRENT_TIME : INT ;
   END_STRUCT ;
   S708 : STRUCT 	//Temporary placeholder variable
    PREVIOUS_TIME : INT ;
    CURRENT_TIME : INT ;
   END_STRUCT ;
   UP_DL : STRUCT 	//Temporary placeholder variable
    PREVIOUS_TIME : INT ;
    CURRENT_TIME : INT ;
   END_STRUCT ;
   IN_TRV : STRUCT 	//Temporary placeholder variable
    PREVIOUS_TIME : INT ;
    CURRENT_TIME : INT ;
   END_STRUCT ;
   SPARE17 : STRUCT 	//Temporary placeholder variable
    PREVIOUS_TIME : INT ;
    CURRENT_TIME : INT ;
   END_STRUCT ;
   SPARE18 : STRUCT 	//Temporary placeholder variable
    PREVIOUS_TIME : INT ;
    CURRENT_TIME : INT ;
   END_STRUCT ;
   SPARE19 : STRUCT 	//Temporary placeholder variable
    PREVIOUS_TIME : INT ;
    CURRENT_TIME : INT ;
   END_STRUCT ;
   SPARE20 : STRUCT 	//Temporary placeholder variable
    PREVIOUS_TIME : INT ;
    CURRENT_TIME : INT ;
   END_STRUCT ;
   SPARE21 : STRUCT 	//Temporary placeholder variable
    PREVIOUS_TIME : INT ;
    CURRENT_TIME : INT ;
   END_STRUCT ;
   SPARE22 : STRUCT 	//Temporary placeholder variable
    PREVIOUS_TIME : INT ;
    CURRENT_TIME : INT ;
   END_STRUCT ;
   SPARE23 : STRUCT 	//Temporary placeholder variable
    PREVIOUS_TIME : INT ;
    CURRENT_TIME : INT ;
   END_STRUCT ;
   SPARE24 : STRUCT 	//Temporary placeholder variable
    PREVIOUS_TIME : INT ;
    CURRENT_TIME : INT ;
   END_STRUCT ;
   SPARE25 : STRUCT 	//Temporary placeholder variable
    PREVIOUS_TIME : INT ;
    CURRENT_TIME : INT ;
   END_STRUCT ;
   SPARE26 : STRUCT 	//Temporary placeholder variable
    PREVIOUS_TIME : INT ;
    CURRENT_TIME : INT ;
   END_STRUCT ;
   ALL_LINE : STRUCT 	//Temporary placeholder variable
    PREVIOUS_TIME : INT ;
    CURRENT_TIME : INT ;
   END_STRUCT ;
   PRODUCT_COUNT_CURRENT : STRUCT 	//Temporary placeholder variable
    COUNT : INT ;
   END_STRUCT ;
   PRODUCT_COUNT_GOAL : STRUCT 	//Temporary placeholder variable
    COUNT : INT ;
   END_STRUCT ;
   SPARE27 : STRUCT 	//Temporary placeholder variable
    PREVIOUS_TIME : INT ;
    CURRENT_TIME : INT ;
   END_STRUCT ;
   SPARE28 : STRUCT 	//Temporary placeholder variable
    PREVIOUS_TIME : INT ;
    CURRENT_TIME : INT ;
   END_STRUCT ;
   SPARE29 : STRUCT 	//Temporary placeholder variable
    PREVIOUS_TIME : INT ;
    CURRENT_TIME : INT ;
   END_STRUCT ;
  END_STRUCT ;
BEGIN
   S700_R1.PREVIOUS_TIME := 0;
   S700_R1.CURRENT_TIME := 0;
   S700_IDLE.PREVIOUS_TIME := 0;
   S700_IDLE.CURRENT_TIME := 0;
   S700_R2.PREVIOUS_TIME := 0;
   S700_R2.CURRENT_TIME := 0;
   S700_1_IDLE.PREVIOUS_TIME := 0;
   S700_1_IDLE.CURRENT_TIME := 0;
   S701_R3.PREVIOUS_TIME := 0;
   S701_R3.CURRENT_TIME := 0;
   S701.PREVIOUS_TIME := 0;
   S701.CURRENT_TIME := 0;
   S701_R4.PREVIOUS_TIME := 0;
   S701_R4.CURRENT_TIME := 0;
   SPARE1.PREVIOUS_TIME := 0;
   SPARE1.CURRENT_TIME := 0;
   SPARE2.PREVIOUS_TIME := 0;
   SPARE2.CURRENT_TIME := 0;
   SPARE3.PREVIOUS_TIME := 0;
   SPARE3.CURRENT_TIME := 0;
   SPARE4.PREVIOUS_TIME := 0;
   SPARE4.CURRENT_TIME := 0;
   SPARE5.PREVIOUS_TIME := 0;
   SPARE5.CURRENT_TIME := 0;
   SPARE6.PREVIOUS_TIME := 0;
   SPARE6.CURRENT_TIME := 0;
   SPARE7.PREVIOUS_TIME := 0;
   SPARE7.CURRENT_TIME := 0;
   SPARE8.PREVIOUS_TIME := 0;
   SPARE8.CURRENT_TIME := 0;
   SPARE9.PREVIOUS_TIME := 0;
   SPARE9.CURRENT_TIME := 0;
   SPARE10.PREVIOUS_TIME := 0;
   SPARE10.CURRENT_TIME := 0;
   SPARE11.PREVIOUS_TIME := 0;
   SPARE11.CURRENT_TIME := 0;
   SPARE12.PREVIOUS_TIME := 0;
   SPARE12.CURRENT_TIME := 0;
   SPARE13.PREVIOUS_TIME := 0;
   SPARE13.CURRENT_TIME := 0;
   SPARE30.PREVIOUS_TIME := 0;
   SPARE30.CURRENT_TIME := 0;
   SPARE31.COUNT := 0;
   SPARE32.COUNT := 0;
   SPARE14.PREVIOUS_TIME := 0;
   SPARE14.CURRENT_TIME := 0;
   SPARE15.PREVIOUS_TIME := 0;
   SPARE15.CURRENT_TIME := 0;
   SPARE16.PREVIOUS_TIME := 0;
   SPARE16.CURRENT_TIME := 0;
   OUT_TRV.PREVIOUS_TIME := 0;
   OUT_TRV.CURRENT_TIME := 0;
   S702.PREVIOUS_TIME := 0;
   S702.CURRENT_TIME := 0;
   S703.PREVIOUS_TIME := 0;
   S703.CURRENT_TIME := 0;
   S704.PREVIOUS_TIME := 0;
   S704.CURRENT_TIME := 0;
   S705.PREVIOUS_TIME := 0;
   S705.CURRENT_TIME := 0;
   S706.PREVIOUS_TIME := 0;
   S706.CURRENT_TIME := 0;
   S707.PREVIOUS_TIME := 0;
   S707.CURRENT_TIME := 0;
   S708.PREVIOUS_TIME := 0;
   S708.CURRENT_TIME := 0;
   UP_DL.PREVIOUS_TIME := 0;
   UP_DL.CURRENT_TIME := 0;
   IN_TRV.PREVIOUS_TIME := 0;
   IN_TRV.CURRENT_TIME := 0;
   SPARE17.PREVIOUS_TIME := 0;
   SPARE17.CURRENT_TIME := 0;
   SPARE18.PREVIOUS_TIME := 0;
   SPARE18.CURRENT_TIME := 0;
   SPARE19.PREVIOUS_TIME := 0;
   SPARE19.CURRENT_TIME := 0;
   SPARE20.PREVIOUS_TIME := 0;
   SPARE20.CURRENT_TIME := 0;
   SPARE21.PREVIOUS_TIME := 0;
   SPARE21.CURRENT_TIME := 0;
   SPARE22.PREVIOUS_TIME := 0;
   SPARE22.CURRENT_TIME := 0;
   SPARE23.PREVIOUS_TIME := 0;
   SPARE23.CURRENT_TIME := 0;
   SPARE24.PREVIOUS_TIME := 0;
   SPARE24.CURRENT_TIME := 0;
   SPARE25.PREVIOUS_TIME := 0;
   SPARE25.CURRENT_TIME := 0;
   SPARE26.PREVIOUS_TIME := 0;
   SPARE26.CURRENT_TIME := 0;
   ALL_LINE.PREVIOUS_TIME := 0;
   ALL_LINE.CURRENT_TIME := 0;
   PRODUCT_COUNT_CURRENT.COUNT := 0;
   PRODUCT_COUNT_GOAL.COUNT := 0;
   SPARE27.PREVIOUS_TIME := 0;
   SPARE27.CURRENT_TIME := 0;
   SPARE28.PREVIOUS_TIME := 0;
   SPARE28.CURRENT_TIME := 0;
   SPARE29.PREVIOUS_TIME := 0;
   SPARE29.CURRENT_TIME := 0;
END_DATA_BLOCK

DATA_BLOCK DB 54
TITLE =
VERSION : 0.1


  STRUCT
   DP_1 : STRUCT 	//Temporary placeholder variable
    CHECK_ACTIVE : BOOL ;
    DATA_FIELD : ARRAY  [0 .. 54 ] OF BYTE ;
    SUM_SLAVE_DIAG : INT ;
    LIST_NOT_PRESENT : ARRAY  [0 .. 3 ] OF DWORD ;
    LIST_ERROR : ARRAY  [0 .. 3 ] OF DWORD ;
    RET_VALUE : INT ;
    DIAG_EVENT : BOOL ;
    STATION_ERR : BOOL ;
    RESTART : BOOL ;
    BUSY : BOOL ;
    SP1 : WORD ;
    SP2 : WORD ;
   END_STRUCT ;
   DP_2 : STRUCT 	//Temporary placeholder variable
    CHECK_ACTIVE : BOOL ;
    DATA_FIELD : ARRAY  [0 .. 54 ] OF BYTE ;
    SUM_SLAVE_DIAG : INT ;
    LIST_NOT_PRESENT : ARRAY  [0 .. 3 ] OF DWORD ;
    LIST_ERROR : ARRAY  [0 .. 3 ] OF DWORD ;
    RET_VALUE : INT ;
    DIAG_EVENT : BOOL ;
    STATION_ERR : BOOL ;
    RESTART : BOOL ;
    BUSY : BOOL ;
    SP1 : WORD ;
    SP2 : WORD ;
   END_STRUCT ;
   DP_3 : STRUCT 	//Temporary placeholder variable
    NDR : BOOL ;
    ERR : BOOL ;
    SP21 : ARRAY  [0 .. 3 ] OF WORD ;
    STATUS : WORD ;
    SP22 : WORD ;
    DIAGLNG : BYTE ;
    SP23 : ARRAY  [0 .. 3 ] OF BYTE ;
    LIST_ERROR : ARRAY  [0 .. 3 ] OF DWORD ;
    SP24 : ARRAY  [0 .. 12 ] OF BYTE ;
   END_STRUCT ;
   DP_4 : STRUCT 	//Temporary placeholder variable
    NDR : BOOL ;
    ERR : BOOL ;
    SP21 : ARRAY  [0 .. 3 ] OF WORD ;
    STATUS : WORD ;
    SP22 : WORD ;
    DIAGLNG : BYTE ;
    SP23 : ARRAY  [0 .. 3 ] OF BYTE ;
    LIST_ERROR : ARRAY  [0 .. 3 ] OF DWORD ;
    SP24 : ARRAY  [0 .. 12 ] OF BYTE ;
   END_STRUCT ;
   DP_5 : STRUCT 	//Temporary placeholder variable
    NDR : BOOL ;
    ERR : BOOL ;
    SP21 : ARRAY  [0 .. 3 ] OF WORD ;
    STATUS : WORD ;
    SP22 : WORD ;
    DIAGLNG : BYTE ;
    SP23 : ARRAY  [0 .. 3 ] OF BYTE ;
    LIST_ERROR : ARRAY  [0 .. 3 ] OF DWORD ;
    SP24 : ARRAY  [0 .. 12 ] OF BYTE ;
   END_STRUCT ;
   DP_6 : STRUCT 	//Temporary placeholder variable
    NDR : BOOL ;
    ERR : BOOL ;
    SP21 : ARRAY  [0 .. 3 ] OF WORD ;
    STATUS : WORD ;
    SP22 : WORD ;
    DIAGLNG : BYTE ;
    SP23 : ARRAY  [0 .. 3 ] OF BYTE ;
    LIST_ERROR : ARRAY  [0 .. 3 ] OF DWORD ;
    SP24 : ARRAY  [0 .. 12 ] OF BYTE ;
   END_STRUCT ;
   DP_7 : STRUCT 	//Temporary placeholder variable
    NDR : BOOL ;
    ERR : BOOL ;
    SP21 : ARRAY  [0 .. 3 ] OF WORD ;
    STATUS : WORD ;
    SP22 : WORD ;
    DIAGLNG : BYTE ;
    SP23 : ARRAY  [0 .. 3 ] OF BYTE ;
    LIST_ERROR : ARRAY  [0 .. 3 ] OF DWORD ;
    SP24 : ARRAY  [0 .. 12 ] OF BYTE ;
   END_STRUCT ;
   DP_8 : STRUCT 	//Temporary placeholder variable
    NDR : BOOL ;
    ERR : BOOL ;
    SP21 : ARRAY  [0 .. 3 ] OF WORD ;
    STATUS : WORD ;
    SP22 : WORD ;
    DIAGLNG : BYTE ;
    SP23 : ARRAY  [0 .. 3 ] OF BYTE ;
    LIST_ERROR : ARRAY  [0 .. 3 ] OF DWORD ;
    SP24 : ARRAY  [0 .. 12 ] OF BYTE ;
   END_STRUCT ;
   DP_9 : STRUCT 	//Temporary placeholder variable
    NDR : BOOL ;
    ERR : BOOL ;
    SP21 : ARRAY  [0 .. 3 ] OF WORD ;
    STATUS : WORD ;
    SP22 : WORD ;
    DIAGLNG : BYTE ;
    SP23 : ARRAY  [0 .. 3 ] OF BYTE ;
    LIST_ERROR : ARRAY  [0 .. 3 ] OF DWORD ;
    SP24 : ARRAY  [0 .. 12 ] OF BYTE ;
   END_STRUCT ;
   DP_10 : STRUCT 	//Temporary placeholder variable
    NDR : BOOL ;
    ERR : BOOL ;
    SP21 : ARRAY  [0 .. 3 ] OF WORD ;
    STATUS : WORD ;
    SP22 : WORD ;
    DIAGLNG : BYTE ;
    SP23 : ARRAY  [0 .. 3 ] OF BYTE ;
    LIST_ERROR : ARRAY  [0 .. 3 ] OF DWORD ;
    SP24 : ARRAY  [0 .. 12 ] OF BYTE ;
   END_STRUCT ;
  END_STRUCT ;
BEGIN
   DP_1.CHECK_ACTIVE := FALSE;
   DP_1.DATA_FIELD[0] := B#16#0;
   DP_1.DATA_FIELD[1] := B#16#0;
   DP_1.DATA_FIELD[2] := B#16#0;
   DP_1.DATA_FIELD[3] := B#16#0;
   DP_1.DATA_FIELD[4] := B#16#0;
   DP_1.DATA_FIELD[5] := B#16#0;
   DP_1.DATA_FIELD[6] := B#16#0;
   DP_1.DATA_FIELD[7] := B#16#0;
   DP_1.DATA_FIELD[8] := B#16#0;
   DP_1.DATA_FIELD[9] := B#16#0;
   DP_1.DATA_FIELD[10] := B#16#0;
   DP_1.DATA_FIELD[11] := B#16#0;
   DP_1.DATA_FIELD[12] := B#16#0;
   DP_1.DATA_FIELD[13] := B#16#0;
   DP_1.DATA_FIELD[14] := B#16#0;
   DP_1.DATA_FIELD[15] := B#16#0;
   DP_1.DATA_FIELD[16] := B#16#0;
   DP_1.DATA_FIELD[17] := B#16#0;
   DP_1.DATA_FIELD[18] := B#16#0;
   DP_1.DATA_FIELD[19] := B#16#0;
   DP_1.DATA_FIELD[20] := B#16#0;
   DP_1.DATA_FIELD[21] := B#16#0;
   DP_1.DATA_FIELD[22] := B#16#0;
   DP_1.DATA_FIELD[23] := B#16#0;
   DP_1.DATA_FIELD[24] := B#16#0;
   DP_1.DATA_FIELD[25] := B#16#0;
   DP_1.DATA_FIELD[26] := B#16#0;
   DP_1.DATA_FIELD[27] := B#16#0;
   DP_1.DATA_FIELD[28] := B#16#0;
   DP_1.DATA_FIELD[29] := B#16#0;
   DP_1.DATA_FIELD[30] := B#16#0;
   DP_1.DATA_FIELD[31] := B#16#0;
   DP_1.DATA_FIELD[32] := B#16#0;
   DP_1.DATA_FIELD[33] := B#16#0;
   DP_1.DATA_FIELD[34] := B#16#0;
   DP_1.DATA_FIELD[35] := B#16#0;
   DP_1.DATA_FIELD[36] := B#16#0;
   DP_1.DATA_FIELD[37] := B#16#0;
   DP_1.DATA_FIELD[38] := B#16#0;
   DP_1.DATA_FIELD[39] := B#16#0;
   DP_1.DATA_FIELD[40] := B#16#0;
   DP_1.DATA_FIELD[41] := B#16#0;
   DP_1.DATA_FIELD[42] := B#16#0;
   DP_1.DATA_FIELD[43] := B#16#0;
   DP_1.DATA_FIELD[44] := B#16#0;
   DP_1.DATA_FIELD[45] := B#16#0;
   DP_1.DATA_FIELD[46] := B#16#0;
   DP_1.DATA_FIELD[47] := B#16#0;
   DP_1.DATA_FIELD[48] := B#16#0;
   DP_1.DATA_FIELD[49] := B#16#0;
   DP_1.DATA_FIELD[50] := B#16#0;
   DP_1.DATA_FIELD[51] := B#16#0;
   DP_1.DATA_FIELD[52] := B#16#0;
   DP_1.DATA_FIELD[53] := B#16#0;
   DP_1.DATA_FIELD[54] := B#16#0;
   DP_1.SUM_SLAVE_DIAG := 0;
   DP_1.LIST_NOT_PRESENT[0] := DW#16#0;
   DP_1.LIST_NOT_PRESENT[1] := DW#16#0;
   DP_1.LIST_NOT_PRESENT[2] := DW#16#0;
   DP_1.LIST_NOT_PRESENT[3] := DW#16#0;
   DP_1.LIST_ERROR[0] := DW#16#0;
   DP_1.LIST_ERROR[1] := DW#16#0;
   DP_1.LIST_ERROR[2] := DW#16#0;
   DP_1.LIST_ERROR[3] := DW#16#0;
   DP_1.RET_VALUE := 0;
   DP_1.DIAG_EVENT := FALSE;
   DP_1.STATION_ERR := FALSE;
   DP_1.RESTART := FALSE;
   DP_1.BUSY := FALSE;
   DP_1.SP1 := W#16#0;
   DP_1.SP2 := W#16#0;
   DP_2.CHECK_ACTIVE := FALSE;
   DP_2.DATA_FIELD[0] := B#16#0;
   DP_2.DATA_FIELD[1] := B#16#0;
   DP_2.DATA_FIELD[2] := B#16#0;
   DP_2.DATA_FIELD[3] := B#16#0;
   DP_2.DATA_FIELD[4] := B#16#0;
   DP_2.DATA_FIELD[5] := B#16#0;
   DP_2.DATA_FIELD[6] := B#16#0;
   DP_2.DATA_FIELD[7] := B#16#0;
   DP_2.DATA_FIELD[8] := B#16#0;
   DP_2.DATA_FIELD[9] := B#16#0;
   DP_2.DATA_FIELD[10] := B#16#0;
   DP_2.DATA_FIELD[11] := B#16#0;
   DP_2.DATA_FIELD[12] := B#16#0;
   DP_2.DATA_FIELD[13] := B#16#0;
   DP_2.DATA_FIELD[14] := B#16#0;
   DP_2.DATA_FIELD[15] := B#16#0;
   DP_2.DATA_FIELD[16] := B#16#0;
   DP_2.DATA_FIELD[17] := B#16#0;
   DP_2.DATA_FIELD[18] := B#16#0;
   DP_2.DATA_FIELD[19] := B#16#0;
   DP_2.DATA_FIELD[20] := B#16#0;
   DP_2.DATA_FIELD[21] := B#16#0;
   DP_2.DATA_FIELD[22] := B#16#0;
   DP_2.DATA_FIELD[23] := B#16#0;
   DP_2.DATA_FIELD[24] := B#16#0;
   DP_2.DATA_FIELD[25] := B#16#0;
   DP_2.DATA_FIELD[26] := B#16#0;
   DP_2.DATA_FIELD[27] := B#16#0;
   DP_2.DATA_FIELD[28] := B#16#0;
   DP_2.DATA_FIELD[29] := B#16#0;
   DP_2.DATA_FIELD[30] := B#16#0;
   DP_2.DATA_FIELD[31] := B#16#0;
   DP_2.DATA_FIELD[32] := B#16#0;
   DP_2.DATA_FIELD[33] := B#16#0;
   DP_2.DATA_FIELD[34] := B#16#0;
   DP_2.DATA_FIELD[35] := B#16#0;
   DP_2.DATA_FIELD[36] := B#16#0;
   DP_2.DATA_FIELD[37] := B#16#0;
   DP_2.DATA_FIELD[38] := B#16#0;
   DP_2.DATA_FIELD[39] := B#16#0;
   DP_2.DATA_FIELD[40] := B#16#0;
   DP_2.DATA_FIELD[41] := B#16#0;
   DP_2.DATA_FIELD[42] := B#16#0;
   DP_2.DATA_FIELD[43] := B#16#0;
   DP_2.DATA_FIELD[44] := B#16#0;
   DP_2.DATA_FIELD[45] := B#16#0;
   DP_2.DATA_FIELD[46] := B#16#0;
   DP_2.DATA_FIELD[47] := B#16#0;
   DP_2.DATA_FIELD[48] := B#16#0;
   DP_2.DATA_FIELD[49] := B#16#0;
   DP_2.DATA_FIELD[50] := B#16#0;
   DP_2.DATA_FIELD[51] := B#16#0;
   DP_2.DATA_FIELD[52] := B#16#0;
   DP_2.DATA_FIELD[53] := B#16#0;
   DP_2.DATA_FIELD[54] := B#16#0;
   DP_2.SUM_SLAVE_DIAG := 0;
   DP_2.LIST_NOT_PRESENT[0] := DW#16#0;
   DP_2.LIST_NOT_PRESENT[1] := DW#16#0;
   DP_2.LIST_NOT_PRESENT[2] := DW#16#0;
   DP_2.LIST_NOT_PRESENT[3] := DW#16#0;
   DP_2.LIST_ERROR[0] := DW#16#0;
   DP_2.LIST_ERROR[1] := DW#16#0;
   DP_2.LIST_ERROR[2] := DW#16#0;
   DP_2.LIST_ERROR[3] := DW#16#0;
   DP_2.RET_VALUE := 0;
   DP_2.DIAG_EVENT := FALSE;
   DP_2.STATION_ERR := FALSE;
   DP_2.RESTART := FALSE;
   DP_2.BUSY := FALSE;
   DP_2.SP1 := W#16#0;
   DP_2.SP2 := W#16#0;
   DP_3.NDR := FALSE;
   DP_3.ERR := FALSE;
   DP_3.SP21[0] := W#16#0;
   DP_3.SP21[1] := W#16#0;
   DP_3.SP21[2] := W#16#0;
   DP_3.SP21[3] := W#16#0;
   DP_3.STATUS := W#16#0;
   DP_3.SP22 := W#16#0;
   DP_3.DIAGLNG := B#16#0;
   DP_3.SP23[0] := B#16#0;
   DP_3.SP23[1] := B#16#0;
   DP_3.SP23[2] := B#16#0;
   DP_3.SP23[3] := B#16#0;
   DP_3.LIST_ERROR[0] := DW#16#0;
   DP_3.LIST_ERROR[1] := DW#16#0;
   DP_3.LIST_ERROR[2] := DW#16#0;
   DP_3.LIST_ERROR[3] := DW#16#0;
   DP_3.SP24[0] := B#16#0;
   DP_3.SP24[1] := B#16#0;
   DP_3.SP24[2] := B#16#0;
   DP_3.SP24[3] := B#16#0;
   DP_3.SP24[4] := B#16#0;
   DP_3.SP24[5] := B#16#0;
   DP_3.SP24[6] := B#16#0;
   DP_3.SP24[7] := B#16#0;
   DP_3.SP24[8] := B#16#0;
   DP_3.SP24[9] := B#16#0;
   DP_3.SP24[10] := B#16#0;
   DP_3.SP24[11] := B#16#0;
   DP_3.SP24[12] := B#16#0;
   DP_4.NDR := FALSE;
   DP_4.ERR := FALSE;
   DP_4.SP21[0] := W#16#0;
   DP_4.SP21[1] := W#16#0;
   DP_4.SP21[2] := W#16#0;
   DP_4.SP21[3] := W#16#0;
   DP_4.STATUS := W#16#0;
   DP_4.SP22 := W#16#0;
   DP_4.DIAGLNG := B#16#0;
   DP_4.SP23[0] := B#16#0;
   DP_4.SP23[1] := B#16#0;
   DP_4.SP23[2] := B#16#0;
   DP_4.SP23[3] := B#16#0;
   DP_4.LIST_ERROR[0] := DW#16#0;
   DP_4.LIST_ERROR[1] := DW#16#0;
   DP_4.LIST_ERROR[2] := DW#16#0;
   DP_4.LIST_ERROR[3] := DW#16#0;
   DP_4.SP24[0] := B#16#0;
   DP_4.SP24[1] := B#16#0;
   DP_4.SP24[2] := B#16#0;
   DP_4.SP24[3] := B#16#0;
   DP_4.SP24[4] := B#16#0;
   DP_4.SP24[5] := B#16#0;
   DP_4.SP24[6] := B#16#0;
   DP_4.SP24[7] := B#16#0;
   DP_4.SP24[8] := B#16#0;
   DP_4.SP24[9] := B#16#0;
   DP_4.SP24[10] := B#16#0;
   DP_4.SP24[11] := B#16#0;
   DP_4.SP24[12] := B#16#0;
   DP_5.NDR := FALSE;
   DP_5.ERR := FALSE;
   DP_5.SP21[0] := W#16#0;
   DP_5.SP21[1] := W#16#0;
   DP_5.SP21[2] := W#16#0;
   DP_5.SP21[3] := W#16#0;
   DP_5.STATUS := W#16#0;
   DP_5.SP22 := W#16#0;
   DP_5.DIAGLNG := B#16#0;
   DP_5.SP23[0] := B#16#0;
   DP_5.SP23[1] := B#16#0;
   DP_5.SP23[2] := B#16#0;
   DP_5.SP23[3] := B#16#0;
   DP_5.LIST_ERROR[0] := DW#16#0;
   DP_5.LIST_ERROR[1] := DW#16#0;
   DP_5.LIST_ERROR[2] := DW#16#0;
   DP_5.LIST_ERROR[3] := DW#16#0;
   DP_5.SP24[0] := B#16#0;
   DP_5.SP24[1] := B#16#0;
   DP_5.SP24[2] := B#16#0;
   DP_5.SP24[3] := B#16#0;
   DP_5.SP24[4] := B#16#0;
   DP_5.SP24[5] := B#16#0;
   DP_5.SP24[6] := B#16#0;
   DP_5.SP24[7] := B#16#0;
   DP_5.SP24[8] := B#16#0;
   DP_5.SP24[9] := B#16#0;
   DP_5.SP24[10] := B#16#0;
   DP_5.SP24[11] := B#16#0;
   DP_5.SP24[12] := B#16#0;
   DP_6.NDR := FALSE;
   DP_6.ERR := FALSE;
   DP_6.SP21[0] := W#16#0;
   DP_6.SP21[1] := W#16#0;
   DP_6.SP21[2] := W#16#0;
   DP_6.SP21[3] := W#16#0;
   DP_6.STATUS := W#16#0;
   DP_6.SP22 := W#16#0;
   DP_6.DIAGLNG := B#16#0;
   DP_6.SP23[0] := B#16#0;
   DP_6.SP23[1] := B#16#0;
   DP_6.SP23[2] := B#16#0;
   DP_6.SP23[3] := B#16#0;
   DP_6.LIST_ERROR[0] := DW#16#0;
   DP_6.LIST_ERROR[1] := DW#16#0;
   DP_6.LIST_ERROR[2] := DW#16#0;
   DP_6.LIST_ERROR[3] := DW#16#0;
   DP_6.SP24[0] := B#16#0;
   DP_6.SP24[1] := B#16#0;
   DP_6.SP24[2] := B#16#0;
   DP_6.SP24[3] := B#16#0;
   DP_6.SP24[4] := B#16#0;
   DP_6.SP24[5] := B#16#0;
   DP_6.SP24[6] := B#16#0;
   DP_6.SP24[7] := B#16#0;
   DP_6.SP24[8] := B#16#0;
   DP_6.SP24[9] := B#16#0;
   DP_6.SP24[10] := B#16#0;
   DP_6.SP24[11] := B#16#0;
   DP_6.SP24[12] := B#16#0;
   DP_7.NDR := FALSE;
   DP_7.ERR := FALSE;
   DP_7.SP21[0] := W#16#0;
   DP_7.SP21[1] := W#16#0;
   DP_7.SP21[2] := W#16#0;
   DP_7.SP21[3] := W#16#0;
   DP_7.STATUS := W#16#0;
   DP_7.SP22 := W#16#0;
   DP_7.DIAGLNG := B#16#0;
   DP_7.SP23[0] := B#16#0;
   DP_7.SP23[1] := B#16#0;
   DP_7.SP23[2] := B#16#0;
   DP_7.SP23[3] := B#16#0;
   DP_7.LIST_ERROR[0] := DW#16#0;
   DP_7.LIST_ERROR[1] := DW#16#0;
   DP_7.LIST_ERROR[2] := DW#16#0;
   DP_7.LIST_ERROR[3] := DW#16#0;
   DP_7.SP24[0] := B#16#0;
   DP_7.SP24[1] := B#16#0;
   DP_7.SP24[2] := B#16#0;
   DP_7.SP24[3] := B#16#0;
   DP_7.SP24[4] := B#16#0;
   DP_7.SP24[5] := B#16#0;
   DP_7.SP24[6] := B#16#0;
   DP_7.SP24[7] := B#16#0;
   DP_7.SP24[8] := B#16#0;
   DP_7.SP24[9] := B#16#0;
   DP_7.SP24[10] := B#16#0;
   DP_7.SP24[11] := B#16#0;
   DP_7.SP24[12] := B#16#0;
   DP_8.NDR := FALSE;
   DP_8.ERR := FALSE;
   DP_8.SP21[0] := W#16#0;
   DP_8.SP21[1] := W#16#0;
   DP_8.SP21[2] := W#16#0;
   DP_8.SP21[3] := W#16#0;
   DP_8.STATUS := W#16#0;
   DP_8.SP22 := W#16#0;
   DP_8.DIAGLNG := B#16#0;
   DP_8.SP23[0] := B#16#0;
   DP_8.SP23[1] := B#16#0;
   DP_8.SP23[2] := B#16#0;
   DP_8.SP23[3] := B#16#0;
   DP_8.LIST_ERROR[0] := DW#16#0;
   DP_8.LIST_ERROR[1] := DW#16#0;
   DP_8.LIST_ERROR[2] := DW#16#0;
   DP_8.LIST_ERROR[3] := DW#16#0;
   DP_8.SP24[0] := B#16#0;
   DP_8.SP24[1] := B#16#0;
   DP_8.SP24[2] := B#16#0;
   DP_8.SP24[3] := B#16#0;
   DP_8.SP24[4] := B#16#0;
   DP_8.SP24[5] := B#16#0;
   DP_8.SP24[6] := B#16#0;
   DP_8.SP24[7] := B#16#0;
   DP_8.SP24[8] := B#16#0;
   DP_8.SP24[9] := B#16#0;
   DP_8.SP24[10] := B#16#0;
   DP_8.SP24[11] := B#16#0;
   DP_8.SP24[12] := B#16#0;
   DP_9.NDR := FALSE;
   DP_9.ERR := FALSE;
   DP_9.SP21[0] := W#16#0;
   DP_9.SP21[1] := W#16#0;
   DP_9.SP21[2] := W#16#0;
   DP_9.SP21[3] := W#16#0;
   DP_9.STATUS := W#16#0;
   DP_9.SP22 := W#16#0;
   DP_9.DIAGLNG := B#16#0;
   DP_9.SP23[0] := B#16#0;
   DP_9.SP23[1] := B#16#0;
   DP_9.SP23[2] := B#16#0;
   DP_9.SP23[3] := B#16#0;
   DP_9.LIST_ERROR[0] := DW#16#0;
   DP_9.LIST_ERROR[1] := DW#16#0;
   DP_9.LIST_ERROR[2] := DW#16#0;
   DP_9.LIST_ERROR[3] := DW#16#0;
   DP_9.SP24[0] := B#16#0;
   DP_9.SP24[1] := B#16#0;
   DP_9.SP24[2] := B#16#0;
   DP_9.SP24[3] := B#16#0;
   DP_9.SP24[4] := B#16#0;
   DP_9.SP24[5] := B#16#0;
   DP_9.SP24[6] := B#16#0;
   DP_9.SP24[7] := B#16#0;
   DP_9.SP24[8] := B#16#0;
   DP_9.SP24[9] := B#16#0;
   DP_9.SP24[10] := B#16#0;
   DP_9.SP24[11] := B#16#0;
   DP_9.SP24[12] := B#16#0;
   DP_10.NDR := FALSE;
   DP_10.ERR := FALSE;
   DP_10.SP21[0] := W#16#0;
   DP_10.SP21[1] := W#16#0;
   DP_10.SP21[2] := W#16#0;
   DP_10.SP21[3] := W#16#0;
   DP_10.STATUS := W#16#0;
   DP_10.SP22 := W#16#0;
   DP_10.DIAGLNG := B#16#0;
   DP_10.SP23[0] := B#16#0;
   DP_10.SP23[1] := B#16#0;
   DP_10.SP23[2] := B#16#0;
   DP_10.SP23[3] := B#16#0;
   DP_10.LIST_ERROR[0] := DW#16#0;
   DP_10.LIST_ERROR[1] := DW#16#0;
   DP_10.LIST_ERROR[2] := DW#16#0;
   DP_10.LIST_ERROR[3] := DW#16#0;
   DP_10.SP24[0] := B#16#0;
   DP_10.SP24[1] := B#16#0;
   DP_10.SP24[2] := B#16#0;
   DP_10.SP24[3] := B#16#0;
   DP_10.SP24[4] := B#16#0;
   DP_10.SP24[5] := B#16#0;
   DP_10.SP24[6] := B#16#0;
   DP_10.SP24[7] := B#16#0;
   DP_10.SP24[8] := B#16#0;
   DP_10.SP24[9] := B#16#0;
   DP_10.SP24[10] := B#16#0;
   DP_10.SP24[11] := B#16#0;
   DP_10.SP24[12] := B#16#0;
END_DATA_BLOCK

DATA_BLOCK DB 55
TITLE =
VERSION : 0.1


  STRUCT
   CP1 : STRUCT
    FC2_NDR : BOOL ;
    FC2_ERROR : BOOL ;
    SP1 : BOOL ;
    SP2 : BOOL ;
    FC1_NDR : BOOL ;
    FC1_ERROR : BOOL ;
    SP3 : BOOL ;
    SP4 : BOOL ;
    FC2_STATUS : WORD ;
    FC2_DPSTATUS : BYTE ;
    FC1_STATUS : WORD ;
    SP5 : WORD ;
    SFC20_1_RET_VAL : INT ;
    SFC20_2_RET_VAL : INT ;
    SFC20_3_RET_VAL : INT ;
    SFC20_4_RET_VAL : INT ;
    SFC20_5_RET_VAL : INT ;
    SFC20_6_RET_VAL : INT ;
    SFC20_7_RET_VAL : INT ;
    SFC20_8_RET_VAL : INT ;
    SFC20_9_RET_VAL : INT ;
    SFC20_10_RET_VAL : INT ;
    SP : ARRAY  [0 .. 9 ] OF WORD ;
   END_STRUCT ;
   CP2 : STRUCT
    FC2_NDR : BOOL ;
    FC2_ERROR : BOOL ;
    SP1 : BOOL ;
    SP2 : BOOL ;
    FC1_NDR : BOOL ;
    FC1_ERROR : BOOL ;
    SP3 : BOOL ;
    SP4 : BOOL ;
    FC2_STATUS : WORD ;
    FC2_DPSTATUS : BYTE ;
    FC1_STATUS : WORD ;
    SP5 : WORD ;
    SFC20_1_RET_VAL : INT ;
    SFC20_2_RET_VAL : INT ;
    SFC20_3_RET_VAL : INT ;
    SFC20_4_RET_VAL : INT ;
    SFC20_5_RET_VAL : INT ;
    SFC20_6_RET_VAL : INT ;
    SFC20_7_RET_VAL : INT ;
    SFC20_8_RET_VAL : INT ;
    SFC20_9_RET_VAL : INT ;
    SFC20_10_RET_VAL : INT ;
    SP : ARRAY  [0 .. 9 ] OF WORD ;
   END_STRUCT ;
   CP3 : STRUCT
    FC2_NDR : BOOL ;
    FC2_ERROR : BOOL ;
    SP1 : BOOL ;
    SP2 : BOOL ;
    FC1_NDR : BOOL ;
    FC1_ERROR : BOOL ;
    SP3 : BOOL ;
    SP4 : BOOL ;
    FC2_STATUS : WORD ;
    FC2_DPSTATUS : BYTE ;
    FC1_STATUS : WORD ;
    SP5 : WORD ;
    SFC20_1_RET_VAL : INT ;
    SFC20_2_RET_VAL : INT ;
    SFC20_3_RET_VAL : INT ;
    SFC20_4_RET_VAL : INT ;
    SFC20_5_RET_VAL : INT ;
    SFC20_6_RET_VAL : INT ;
    SFC20_7_RET_VAL : INT ;
    SFC20_8_RET_VAL : INT ;
    SFC20_9_RET_VAL : INT ;
    SFC20_10_RET_VAL : INT ;
    SP : ARRAY  [0 .. 9 ] OF WORD ;
   END_STRUCT ;
   CP4 : STRUCT
    FC2_NDR : BOOL ;
    FC2_ERROR : BOOL ;
    SP1 : BOOL ;
    SP2 : BOOL ;
    FC1_NDR : BOOL ;
    FC1_ERROR : BOOL ;
    SP3 : BOOL ;
    SP4 : BOOL ;
    FC2_STATUS : WORD ;
    FC2_DPSTATUS : BYTE ;
    FC1_STATUS : WORD ;
    SP5 : WORD ;
    SFC20_1_RET_VAL : INT ;
    SFC20_2_RET_VAL : INT ;
    SFC20_3_RET_VAL : INT ;
    SFC20_4_RET_VAL : INT ;
    SFC20_5_RET_VAL : INT ;
    SFC20_6_RET_VAL : INT ;
    SFC20_7_RET_VAL : INT ;
    SFC20_8_RET_VAL : INT ;
    SFC20_9_RET_VAL : INT ;
    SFC20_10_RET_VAL : INT ;
    SP : ARRAY  [0 .. 9 ] OF WORD ;
   END_STRUCT ;
   CP5 : STRUCT
    FC2_NDR : BOOL ;
    FC2_ERROR : BOOL ;
    SP1 : BOOL ;
    SP2 : BOOL ;
    FC1_NDR : BOOL ;
    FC1_ERROR : BOOL ;
    SP3 : BOOL ;
    SP4 : BOOL ;
    FC2_STATUS : WORD ;
    FC2_DPSTATUS : BYTE ;
    FC1_STATUS : WORD ;
    SP5 : WORD ;
    SFC20_1_RET_VAL : INT ;
    SFC20_2_RET_VAL : INT ;
    SFC20_3_RET_VAL : INT ;
    SFC20_4_RET_VAL : INT ;
    SFC20_5_RET_VAL : INT ;
    SFC20_6_RET_VAL : INT ;
    SFC20_7_RET_VAL : INT ;
    SFC20_8_RET_VAL : INT ;
    SFC20_9_RET_VAL : INT ;
    SFC20_10_RET_VAL : INT ;
    SP : ARRAY  [0 .. 9 ] OF WORD ;
   END_STRUCT ;
   CP6 : STRUCT
    FC2_NDR : BOOL ;
    FC2_ERROR : BOOL ;
    SP1 : BOOL ;
    SP2 : BOOL ;
    FC1_NDR : BOOL ;
    FC1_ERROR : BOOL ;
    SP3 : BOOL ;
    SP4 : BOOL ;
    FC2_STATUS : WORD ;
    FC2_DPSTATUS : BYTE ;
    FC1_STATUS : WORD ;
    SP5 : WORD ;
    SFC20_1_RET_VAL : INT ;
    SFC20_2_RET_VAL : INT ;
    SFC20_3_RET_VAL : INT ;
    SFC20_4_RET_VAL : INT ;
    SFC20_5_RET_VAL : INT ;
    SFC20_6_RET_VAL : INT ;
    SFC20_7_RET_VAL : INT ;
    SFC20_8_RET_VAL : INT ;
    SFC20_9_RET_VAL : INT ;
    SFC20_10_RET_VAL : INT ;
    SP : ARRAY  [0 .. 9 ] OF WORD ;
   END_STRUCT ;
   CP7 : STRUCT
    FC2_NDR : BOOL ;
    FC2_ERROR : BOOL ;
    SP1 : BOOL ;
    SP2 : BOOL ;
    FC1_NDR : BOOL ;
    FC1_ERROR : BOOL ;
    SP3 : BOOL ;
    SP4 : BOOL ;
    FC2_STATUS : WORD ;
    FC2_DPSTATUS : BYTE ;
    FC1_STATUS : WORD ;
    SP5 : WORD ;
    SFC20_1_RET_VAL : INT ;
    SFC20_2_RET_VAL : INT ;
    SFC20_3_RET_VAL : INT ;
    SFC20_4_RET_VAL : INT ;
    SFC20_5_RET_VAL : INT ;
    SFC20_6_RET_VAL : INT ;
    SFC20_7_RET_VAL : INT ;
    SFC20_8_RET_VAL : INT ;
    SFC20_9_RET_VAL : INT ;
    SFC20_10_RET_VAL : INT ;
    SP : ARRAY  [0 .. 9 ] OF WORD ;
   END_STRUCT ;
   CP8 : STRUCT
    FC2_NDR : BOOL ;
    FC2_ERROR : BOOL ;
    SP1 : BOOL ;
    SP2 : BOOL ;
    FC1_NDR : BOOL ;
    FC1_ERROR : BOOL ;
    SP3 : BOOL ;
    SP4 : BOOL ;
    FC2_STATUS : WORD ;
    FC2_DPSTATUS : BYTE ;
    FC1_STATUS : WORD ;
    SP5 : WORD ;
    SFC20_1_RET_VAL : INT ;
    SFC20_2_RET_VAL : INT ;
    SFC20_3_RET_VAL : INT ;
    SFC20_4_RET_VAL : INT ;
    SFC20_5_RET_VAL : INT ;
    SFC20_6_RET_VAL : INT ;
    SFC20_7_RET_VAL : INT ;
    SFC20_8_RET_VAL : INT ;
    SFC20_9_RET_VAL : INT ;
    SFC20_10_RET_VAL : INT ;
    SP : ARRAY  [0 .. 9 ] OF WORD ;
   END_STRUCT ;
   RTN_VALUE_WORD : ARRAY  [0 .. 49 ] OF WORD ;
   AG1 : STRUCT
    FC6_NDR : BOOL ;
    FC6_ERROR : BOOL ;
    SP1 : BOOL ;
    SP2 : BOOL ;
    FC5_NDR : BOOL ;
    FC5_ERROR : BOOL ;
    SP3 : BOOL ;
    SP4 : BOOL ;
    FC6_STATUS : WORD ;
    FC6_DPSTATUS : BYTE ;
    FC5_STATUS : WORD ;
    SP5 : WORD ;
    SFC20_1_RET_VAL : INT ;
    SFC20_2_RET_VAL : INT ;
    SFC20_3_RET_VAL : INT ;
    SFC20_4_RET_VAL : INT ;
    SFC20_5_RET_VAL : INT ;
    SFC20_6_RET_VAL : INT ;
    SFC20_7_RET_VAL : INT ;
    SFC20_8_RET_VAL : INT ;
    SFC20_9_RET_VAL : INT ;
    SFC20_10_RET_VAL : INT ;
    SP : ARRAY  [0 .. 9 ] OF WORD ;
   END_STRUCT ;
   AG2 : STRUCT
    FC6_NDR : BOOL ;
    FC6_ERROR : BOOL ;
    SP1 : BOOL ;
    SP2 : BOOL ;
    FC5_NDR : BOOL ;
    FC5_ERROR : BOOL ;
    SP3 : BOOL ;
    SP4 : BOOL ;
    FC6_STATUS : WORD ;
    FC6_DPSTATUS : BYTE ;
    FC5_STATUS : WORD ;
    SP5 : WORD ;
    SFC20_1_RET_VAL : INT ;
    SFC20_2_RET_VAL : INT ;
    SFC20_3_RET_VAL : INT ;
    SFC20_4_RET_VAL : INT ;
    SFC20_5_RET_VAL : INT ;
    SFC20_6_RET_VAL : INT ;
    SFC20_7_RET_VAL : INT ;
    SFC20_8_RET_VAL : INT ;
    SFC20_9_RET_VAL : INT ;
    SFC20_10_RET_VAL : INT ;
    SP : ARRAY  [0 .. 9 ] OF WORD ;
   END_STRUCT ;
   AG3 : STRUCT
    FC6_NDR : BOOL ;
    FC6_ERROR : BOOL ;
    SP1 : BOOL ;
    SP2 : BOOL ;
    FC5_NDR : BOOL ;
    FC5_ERROR : BOOL ;
    SP3 : BOOL ;
    SP4 : BOOL ;
    FC6_STATUS : WORD ;
    FC6_DPSTATUS : BYTE ;
    FC5_STATUS : WORD ;
    SP5 : WORD ;
    SFC20_1_RET_VAL : INT ;
    SFC20_2_RET_VAL : INT ;
    SFC20_3_RET_VAL : INT ;
    SFC20_4_RET_VAL : INT ;
    SFC20_5_RET_VAL : INT ;
    SFC20_6_RET_VAL : INT ;
    SFC20_7_RET_VAL : INT ;
    SFC20_8_RET_VAL : INT ;
    SFC20_9_RET_VAL : INT ;
    SFC20_10_RET_VAL : INT ;
    SP : ARRAY  [0 .. 9 ] OF WORD ;
   END_STRUCT ;
   AG4 : STRUCT
    FC6_NDR : BOOL ;
    FC6_ERROR : BOOL ;
    SP1 : BOOL ;
    SP2 : BOOL ;
    FC5_NDR : BOOL ;
    FC5_ERROR : BOOL ;
    SP3 : BOOL ;
    SP4 : BOOL ;
    FC6_STATUS : WORD ;
    FC6_DPSTATUS : BYTE ;
    FC5_STATUS : WORD ;
    SP5 : WORD ;
    SFC20_1_RET_VAL : INT ;
    SFC20_2_RET_VAL : INT ;
    SFC20_3_RET_VAL : INT ;
    SFC20_4_RET_VAL : INT ;
    SFC20_5_RET_VAL : INT ;
    SFC20_6_RET_VAL : INT ;
    SFC20_7_RET_VAL : INT ;
    SFC20_8_RET_VAL : INT ;
    SFC20_9_RET_VAL : INT ;
    SFC20_10_RET_VAL : INT ;
    SP : ARRAY  [0 .. 9 ] OF WORD ;
   END_STRUCT ;
   AG5 : STRUCT
    FC6_NDR : BOOL ;
    FC6_ERROR : BOOL ;
    SP1 : BOOL ;
    SP2 : BOOL ;
    FC5_NDR : BOOL ;
    FC5_ERROR : BOOL ;
    SP3 : BOOL ;
    SP4 : BOOL ;
    FC6_STATUS : WORD ;
    FC6_DPSTATUS : BYTE ;
    FC5_STATUS : WORD ;
    SP5 : WORD ;
    SFC20_1_RET_VAL : INT ;
    SFC20_2_RET_VAL : INT ;
    SFC20_3_RET_VAL : INT ;
    SFC20_4_RET_VAL : INT ;
    SFC20_5_RET_VAL : INT ;
    SFC20_6_RET_VAL : INT ;
    SFC20_7_RET_VAL : INT ;
    SFC20_8_RET_VAL : INT ;
    SFC20_9_RET_VAL : INT ;
    SFC20_10_RET_VAL : INT ;
    SP : ARRAY  [0 .. 9 ] OF WORD ;
   END_STRUCT ;
   AG6 : STRUCT
    FC6_NDR : BOOL ;
    FC6_ERROR : BOOL ;
    SP1 : BOOL ;
    SP2 : BOOL ;
    FC5_NDR : BOOL ;
    FC5_ERROR : BOOL ;
    SP3 : BOOL ;
    SP4 : BOOL ;
    FC6_STATUS : WORD ;
    FC6_DPSTATUS : BYTE ;
    FC5_STATUS : WORD ;
    SP5 : WORD ;
    SFC20_1_RET_VAL : INT ;
    SFC20_2_RET_VAL : INT ;
    SFC20_3_RET_VAL : INT ;
    SFC20_4_RET_VAL : INT ;
    SFC20_5_RET_VAL : INT ;
    SFC20_6_RET_VAL : INT ;
    SFC20_7_RET_VAL : INT ;
    SFC20_8_RET_VAL : INT ;
    SFC20_9_RET_VAL : INT ;
    SFC20_10_RET_VAL : INT ;
    SP : ARRAY  [0 .. 9 ] OF WORD ;
   END_STRUCT ;
   AG7 : STRUCT
    FC6_NDR : BOOL ;
    FC6_ERROR : BOOL ;
    SP1 : BOOL ;
    SP2 : BOOL ;
    FC5_NDR : BOOL ;
    FC5_ERROR : BOOL ;
    SP3 : BOOL ;
    SP4 : BOOL ;
    FC6_STATUS : WORD ;
    FC6_DPSTATUS : BYTE ;
    FC5_STATUS : WORD ;
    SP5 : WORD ;
    SFC20_1_RET_VAL : INT ;
    SFC20_2_RET_VAL : INT ;
    SFC20_3_RET_VAL : INT ;
    SFC20_4_RET_VAL : INT ;
    SFC20_5_RET_VAL : INT ;
    SFC20_6_RET_VAL : INT ;
    SFC20_7_RET_VAL : INT ;
    SFC20_8_RET_VAL : INT ;
    SFC20_9_RET_VAL : INT ;
    SFC20_10_RET_VAL : INT ;
    SP : ARRAY  [0 .. 9 ] OF WORD ;
   END_STRUCT ;
   SP : ARRAY  [0 .. 74 ] OF WORD ;
   CTYPE_RET_VAL : ARRAY  [0 .. 99 ] OF INT ;
   MES_RET_VAL1 : ARRAY  [0 .. 199 ] OF INT ;
  END_STRUCT ;
BEGIN
   CP1.FC2_NDR := FALSE;
   CP1.FC2_ERROR := FALSE;
   CP1.SP1 := FALSE;
   CP1.SP2 := FALSE;
   CP1.FC1_NDR := FALSE;
   CP1.FC1_ERROR := FALSE;
   CP1.SP3 := FALSE;
   CP1.SP4 := FALSE;
   CP1.FC2_STATUS := W#16#0;
   CP1.FC2_DPSTATUS := B#16#0;
   CP1.FC1_STATUS := W#16#0;
   CP1.SP5 := W#16#0;
   CP1.SFC20_1_RET_VAL := 0;
   CP1.SFC20_2_RET_VAL := 0;
   CP1.SFC20_3_RET_VAL := 0;
   CP1.SFC20_4_RET_VAL := 0;
   CP1.SFC20_5_RET_VAL := 0;
   CP1.SFC20_6_RET_VAL := 0;
   CP1.SFC20_7_RET_VAL := 0;
   CP1.SFC20_8_RET_VAL := 0;
   CP1.SFC20_9_RET_VAL := 0;
   CP1.SFC20_10_RET_VAL := 0;
   CP1.SP[0] := W#16#0;
   CP1.SP[1] := W#16#0;
   CP1.SP[2] := W#16#0;
   CP1.SP[3] := W#16#0;
   CP1.SP[4] := W#16#0;
   CP1.SP[5] := W#16#0;
   CP1.SP[6] := W#16#0;
   CP1.SP[7] := W#16#0;
   CP1.SP[8] := W#16#0;
   CP1.SP[9] := W#16#0;
   CP2.FC2_NDR := FALSE;
   CP2.FC2_ERROR := FALSE;
   CP2.SP1 := FALSE;
   CP2.SP2 := FALSE;
   CP2.FC1_NDR := FALSE;
   CP2.FC1_ERROR := FALSE;
   CP2.SP3 := FALSE;
   CP2.SP4 := FALSE;
   CP2.FC2_STATUS := W#16#0;
   CP2.FC2_DPSTATUS := B#16#0;
   CP2.FC1_STATUS := W#16#0;
   CP2.SP5 := W#16#0;
   CP2.SFC20_1_RET_VAL := 0;
   CP2.SFC20_2_RET_VAL := 0;
   CP2.SFC20_3_RET_VAL := 0;
   CP2.SFC20_4_RET_VAL := 0;
   CP2.SFC20_5_RET_VAL := 0;
   CP2.SFC20_6_RET_VAL := 0;
   CP2.SFC20_7_RET_VAL := 0;
   CP2.SFC20_8_RET_VAL := 0;
   CP2.SFC20_9_RET_VAL := 0;
   CP2.SFC20_10_RET_VAL := 0;
   CP2.SP[0] := W#16#0;
   CP2.SP[1] := W#16#0;
   CP2.SP[2] := W#16#0;
   CP2.SP[3] := W#16#0;
   CP2.SP[4] := W#16#0;
   CP2.SP[5] := W#16#0;
   CP2.SP[6] := W#16#0;
   CP2.SP[7] := W#16#0;
   CP2.SP[8] := W#16#0;
   CP2.SP[9] := W#16#0;
   CP3.FC2_NDR := FALSE;
   CP3.FC2_ERROR := FALSE;
   CP3.SP1 := FALSE;
   CP3.SP2 := FALSE;
   CP3.FC1_NDR := FALSE;
   CP3.FC1_ERROR := FALSE;
   CP3.SP3 := FALSE;
   CP3.SP4 := FALSE;
   CP3.FC2_STATUS := W#16#0;
   CP3.FC2_DPSTATUS := B#16#0;
   CP3.FC1_STATUS := W#16#0;
   CP3.SP5 := W#16#0;
   CP3.SFC20_1_RET_VAL := 0;
   CP3.SFC20_2_RET_VAL := 0;
   CP3.SFC20_3_RET_VAL := 0;
   CP3.SFC20_4_RET_VAL := 0;
   CP3.SFC20_5_RET_VAL := 0;
   CP3.SFC20_6_RET_VAL := 0;
   CP3.SFC20_7_RET_VAL := 0;
   CP3.SFC20_8_RET_VAL := 0;
   CP3.SFC20_9_RET_VAL := 0;
   CP3.SFC20_10_RET_VAL := 0;
   CP3.SP[0] := W#16#0;
   CP3.SP[1] := W#16#0;
   CP3.SP[2] := W#16#0;
   CP3.SP[3] := W#16#0;
   CP3.SP[4] := W#16#0;
   CP3.SP[5] := W#16#0;
   CP3.SP[6] := W#16#0;
   CP3.SP[7] := W#16#0;
   CP3.SP[8] := W#16#0;
   CP3.SP[9] := W#16#0;
   CP4.FC2_NDR := FALSE;
   CP4.FC2_ERROR := FALSE;
   CP4.SP1 := FALSE;
   CP4.SP2 := FALSE;
   CP4.FC1_NDR := FALSE;
   CP4.FC1_ERROR := FALSE;
   CP4.SP3 := FALSE;
   CP4.SP4 := FALSE;
   CP4.FC2_STATUS := W#16#0;
   CP4.FC2_DPSTATUS := B#16#0;
   CP4.FC1_STATUS := W#16#0;
   CP4.SP5 := W#16#0;
   CP4.SFC20_1_RET_VAL := 0;
   CP4.SFC20_2_RET_VAL := 0;
   CP4.SFC20_3_RET_VAL := 0;
   CP4.SFC20_4_RET_VAL := 0;
   CP4.SFC20_5_RET_VAL := 0;
   CP4.SFC20_6_RET_VAL := 0;
   CP4.SFC20_7_RET_VAL := 0;
   CP4.SFC20_8_RET_VAL := 0;
   CP4.SFC20_9_RET_VAL := 0;
   CP4.SFC20_10_RET_VAL := 0;
   CP4.SP[0] := W#16#0;
   CP4.SP[1] := W#16#0;
   CP4.SP[2] := W#16#0;
   CP4.SP[3] := W#16#0;
   CP4.SP[4] := W#16#0;
   CP4.SP[5] := W#16#0;
   CP4.SP[6] := W#16#0;
   CP4.SP[7] := W#16#0;
   CP4.SP[8] := W#16#0;
   CP4.SP[9] := W#16#0;
   CP5.FC2_NDR := FALSE;
   CP5.FC2_ERROR := FALSE;
   CP5.SP1 := FALSE;
   CP5.SP2 := FALSE;
   CP5.FC1_NDR := FALSE;
   CP5.FC1_ERROR := FALSE;
   CP5.SP3 := FALSE;
   CP5.SP4 := FALSE;
   CP5.FC2_STATUS := W#16#0;
   CP5.FC2_DPSTATUS := B#16#0;
   CP5.FC1_STATUS := W#16#0;
   CP5.SP5 := W#16#0;
   CP5.SFC20_1_RET_VAL := 0;
   CP5.SFC20_2_RET_VAL := 0;
   CP5.SFC20_3_RET_VAL := 0;
   CP5.SFC20_4_RET_VAL := 0;
   CP5.SFC20_5_RET_VAL := 0;
   CP5.SFC20_6_RET_VAL := 0;
   CP5.SFC20_7_RET_VAL := 0;
   CP5.SFC20_8_RET_VAL := 0;
   CP5.SFC20_9_RET_VAL := 0;
   CP5.SFC20_10_RET_VAL := 0;
   CP5.SP[0] := W#16#0;
   CP5.SP[1] := W#16#0;
   CP5.SP[2] := W#16#0;
   CP5.SP[3] := W#16#0;
   CP5.SP[4] := W#16#0;
   CP5.SP[5] := W#16#0;
   CP5.SP[6] := W#16#0;
   CP5.SP[7] := W#16#0;
   CP5.SP[8] := W#16#0;
   CP5.SP[9] := W#16#0;
   CP6.FC2_NDR := FALSE;
   CP6.FC2_ERROR := FALSE;
   CP6.SP1 := FALSE;
   CP6.SP2 := FALSE;
   CP6.FC1_NDR := FALSE;
   CP6.FC1_ERROR := FALSE;
   CP6.SP3 := FALSE;
   CP6.SP4 := FALSE;
   CP6.FC2_STATUS := W#16#0;
   CP6.FC2_DPSTATUS := B#16#0;
   CP6.FC1_STATUS := W#16#0;
   CP6.SP5 := W#16#0;
   CP6.SFC20_1_RET_VAL := 0;
   CP6.SFC20_2_RET_VAL := 0;
   CP6.SFC20_3_RET_VAL := 0;
   CP6.SFC20_4_RET_VAL := 0;
   CP6.SFC20_5_RET_VAL := 0;
   CP6.SFC20_6_RET_VAL := 0;
   CP6.SFC20_7_RET_VAL := 0;
   CP6.SFC20_8_RET_VAL := 0;
   CP6.SFC20_9_RET_VAL := 0;
   CP6.SFC20_10_RET_VAL := 0;
   CP6.SP[0] := W#16#0;
   CP6.SP[1] := W#16#0;
   CP6.SP[2] := W#16#0;
   CP6.SP[3] := W#16#0;
   CP6.SP[4] := W#16#0;
   CP6.SP[5] := W#16#0;
   CP6.SP[6] := W#16#0;
   CP6.SP[7] := W#16#0;
   CP6.SP[8] := W#16#0;
   CP6.SP[9] := W#16#0;
   CP7.FC2_NDR := FALSE;
   CP7.FC2_ERROR := FALSE;
   CP7.SP1 := FALSE;
   CP7.SP2 := FALSE;
   CP7.FC1_NDR := FALSE;
   CP7.FC1_ERROR := FALSE;
   CP7.SP3 := FALSE;
   CP7.SP4 := FALSE;
   CP7.FC2_STATUS := W#16#0;
   CP7.FC2_DPSTATUS := B#16#0;
   CP7.FC1_STATUS := W#16#0;
   CP7.SP5 := W#16#0;
   CP7.SFC20_1_RET_VAL := 0;
   CP7.SFC20_2_RET_VAL := 0;
   CP7.SFC20_3_RET_VAL := 0;
   CP7.SFC20_4_RET_VAL := 0;
   CP7.SFC20_5_RET_VAL := 0;
   CP7.SFC20_6_RET_VAL := 0;
   CP7.SFC20_7_RET_VAL := 0;
   CP7.SFC20_8_RET_VAL := 0;
   CP7.SFC20_9_RET_VAL := 0;
   CP7.SFC20_10_RET_VAL := 0;
   CP7.SP[0] := W#16#0;
   CP7.SP[1] := W#16#0;
   CP7.SP[2] := W#16#0;
   CP7.SP[3] := W#16#0;
   CP7.SP[4] := W#16#0;
   CP7.SP[5] := W#16#0;
   CP7.SP[6] := W#16#0;
   CP7.SP[7] := W#16#0;
   CP7.SP[8] := W#16#0;
   CP7.SP[9] := W#16#0;
   CP8.FC2_NDR := FALSE;
   CP8.FC2_ERROR := FALSE;
   CP8.SP1 := FALSE;
   CP8.SP2 := FALSE;
   CP8.FC1_NDR := FALSE;
   CP8.FC1_ERROR := FALSE;
   CP8.SP3 := FALSE;
   CP8.SP4 := FALSE;
   CP8.FC2_STATUS := W#16#0;
   CP8.FC2_DPSTATUS := B#16#0;
   CP8.FC1_STATUS := W#16#0;
   CP8.SP5 := W#16#0;
   CP8.SFC20_1_RET_VAL := 0;
   CP8.SFC20_2_RET_VAL := 0;
   CP8.SFC20_3_RET_VAL := 0;
   CP8.SFC20_4_RET_VAL := 0;
   CP8.SFC20_5_RET_VAL := 0;
   CP8.SFC20_6_RET_VAL := 0;
   CP8.SFC20_7_RET_VAL := 0;
   CP8.SFC20_8_RET_VAL := 0;
   CP8.SFC20_9_RET_VAL := 0;
   CP8.SFC20_10_RET_VAL := 0;
   CP8.SP[0] := W#16#0;
   CP8.SP[1] := W#16#0;
   CP8.SP[2] := W#16#0;
   CP8.SP[3] := W#16#0;
   CP8.SP[4] := W#16#0;
   CP8.SP[5] := W#16#0;
   CP8.SP[6] := W#16#0;
   CP8.SP[7] := W#16#0;
   CP8.SP[8] := W#16#0;
   CP8.SP[9] := W#16#0;
   RTN_VALUE_WORD[0] := W#16#0;
   RTN_VALUE_WORD[1] := W#16#0;
   RTN_VALUE_WORD[2] := W#16#0;
   RTN_VALUE_WORD[3] := W#16#0;
   RTN_VALUE_WORD[4] := W#16#0;
   RTN_VALUE_WORD[5] := W#16#0;
   RTN_VALUE_WORD[6] := W#16#0;
   RTN_VALUE_WORD[7] := W#16#0;
   RTN_VALUE_WORD[8] := W#16#0;
   RTN_VALUE_WORD[9] := W#16#0;
   RTN_VALUE_WORD[10] := W#16#0;
   RTN_VALUE_WORD[11] := W#16#0;
   RTN_VALUE_WORD[12] := W#16#0;
   RTN_VALUE_WORD[13] := W#16#0;
   RTN_VALUE_WORD[14] := W#16#0;
   RTN_VALUE_WORD[15] := W#16#0;
   RTN_VALUE_WORD[16] := W#16#0;
   RTN_VALUE_WORD[17] := W#16#0;
   RTN_VALUE_WORD[18] := W#16#0;
   RTN_VALUE_WORD[19] := W#16#0;
   RTN_VALUE_WORD[20] := W#16#0;
   RTN_VALUE_WORD[21] := W#16#0;
   RTN_VALUE_WORD[22] := W#16#0;
   RTN_VALUE_WORD[23] := W#16#0;
   RTN_VALUE_WORD[24] := W#16#0;
   RTN_VALUE_WORD[25] := W#16#0;
   RTN_VALUE_WORD[26] := W#16#0;
   RTN_VALUE_WORD[27] := W#16#0;
   RTN_VALUE_WORD[28] := W#16#0;
   RTN_VALUE_WORD[29] := W#16#0;
   RTN_VALUE_WORD[30] := W#16#0;
   RTN_VALUE_WORD[31] := W#16#0;
   RTN_VALUE_WORD[32] := W#16#0;
   RTN_VALUE_WORD[33] := W#16#0;
   RTN_VALUE_WORD[34] := W#16#0;
   RTN_VALUE_WORD[35] := W#16#0;
   RTN_VALUE_WORD[36] := W#16#0;
   RTN_VALUE_WORD[37] := W#16#0;
   RTN_VALUE_WORD[38] := W#16#0;
   RTN_VALUE_WORD[39] := W#16#0;
   RTN_VALUE_WORD[40] := W#16#0;
   RTN_VALUE_WORD[41] := W#16#0;
   RTN_VALUE_WORD[42] := W#16#0;
   RTN_VALUE_WORD[43] := W#16#0;
   RTN_VALUE_WORD[44] := W#16#0;
   RTN_VALUE_WORD[45] := W#16#0;
   RTN_VALUE_WORD[46] := W#16#0;
   RTN_VALUE_WORD[47] := W#16#0;
   RTN_VALUE_WORD[48] := W#16#0;
   RTN_VALUE_WORD[49] := W#16#0;
   AG1.FC6_NDR := FALSE;
   AG1.FC6_ERROR := FALSE;
   AG1.SP1 := FALSE;
   AG1.SP2 := FALSE;
   AG1.FC5_NDR := FALSE;
   AG1.FC5_ERROR := FALSE;
   AG1.SP3 := FALSE;
   AG1.SP4 := FALSE;
   AG1.FC6_STATUS := W#16#0;
   AG1.FC6_DPSTATUS := B#16#0;
   AG1.FC5_STATUS := W#16#0;
   AG1.SP5 := W#16#0;
   AG1.SFC20_1_RET_VAL := 0;
   AG1.SFC20_2_RET_VAL := 0;
   AG1.SFC20_3_RET_VAL := 0;
   AG1.SFC20_4_RET_VAL := 0;
   AG1.SFC20_5_RET_VAL := 0;
   AG1.SFC20_6_RET_VAL := 0;
   AG1.SFC20_7_RET_VAL := 0;
   AG1.SFC20_8_RET_VAL := 0;
   AG1.SFC20_9_RET_VAL := 0;
   AG1.SFC20_10_RET_VAL := 0;
   AG1.SP[0] := W#16#0;
   AG1.SP[1] := W#16#0;
   AG1.SP[2] := W#16#0;
   AG1.SP[3] := W#16#0;
   AG1.SP[4] := W#16#0;
   AG1.SP[5] := W#16#0;
   AG1.SP[6] := W#16#0;
   AG1.SP[7] := W#16#0;
   AG1.SP[8] := W#16#0;
   AG1.SP[9] := W#16#0;
   AG2.FC6_NDR := FALSE;
   AG2.FC6_ERROR := FALSE;
   AG2.SP1 := FALSE;
   AG2.SP2 := FALSE;
   AG2.FC5_NDR := FALSE;
   AG2.FC5_ERROR := FALSE;
   AG2.SP3 := FALSE;
   AG2.SP4 := FALSE;
   AG2.FC6_STATUS := W#16#0;
   AG2.FC6_DPSTATUS := B#16#0;
   AG2.FC5_STATUS := W#16#0;
   AG2.SP5 := W#16#0;
   AG2.SFC20_1_RET_VAL := 0;
   AG2.SFC20_2_RET_VAL := 0;
   AG2.SFC20_3_RET_VAL := 0;
   AG2.SFC20_4_RET_VAL := 0;
   AG2.SFC20_5_RET_VAL := 0;
   AG2.SFC20_6_RET_VAL := 0;
   AG2.SFC20_7_RET_VAL := 0;
   AG2.SFC20_8_RET_VAL := 0;
   AG2.SFC20_9_RET_VAL := 0;
   AG2.SFC20_10_RET_VAL := 0;
   AG2.SP[0] := W#16#0;
   AG2.SP[1] := W#16#0;
   AG2.SP[2] := W#16#0;
   AG2.SP[3] := W#16#0;
   AG2.SP[4] := W#16#0;
   AG2.SP[5] := W#16#0;
   AG2.SP[6] := W#16#0;
   AG2.SP[7] := W#16#0;
   AG2.SP[8] := W#16#0;
   AG2.SP[9] := W#16#0;
   AG3.FC6_NDR := FALSE;
   AG3.FC6_ERROR := FALSE;
   AG3.SP1 := FALSE;
   AG3.SP2 := FALSE;
   AG3.FC5_NDR := FALSE;
   AG3.FC5_ERROR := FALSE;
   AG3.SP3 := FALSE;
   AG3.SP4 := FALSE;
   AG3.FC6_STATUS := W#16#0;
   AG3.FC6_DPSTATUS := B#16#0;
   AG3.FC5_STATUS := W#16#0;
   AG3.SP5 := W#16#0;
   AG3.SFC20_1_RET_VAL := 0;
   AG3.SFC20_2_RET_VAL := 0;
   AG3.SFC20_3_RET_VAL := 0;
   AG3.SFC20_4_RET_VAL := 0;
   AG3.SFC20_5_RET_VAL := 0;
   AG3.SFC20_6_RET_VAL := 0;
   AG3.SFC20_7_RET_VAL := 0;
   AG3.SFC20_8_RET_VAL := 0;
   AG3.SFC20_9_RET_VAL := 0;
   AG3.SFC20_10_RET_VAL := 0;
   AG3.SP[0] := W#16#0;
   AG3.SP[1] := W#16#0;
   AG3.SP[2] := W#16#0;
   AG3.SP[3] := W#16#0;
   AG3.SP[4] := W#16#0;
   AG3.SP[5] := W#16#0;
   AG3.SP[6] := W#16#0;
   AG3.SP[7] := W#16#0;
   AG3.SP[8] := W#16#0;
   AG3.SP[9] := W#16#0;
   AG4.FC6_NDR := FALSE;
   AG4.FC6_ERROR := FALSE;
   AG4.SP1 := FALSE;
   AG4.SP2 := FALSE;
   AG4.FC5_NDR := FALSE;
   AG4.FC5_ERROR := FALSE;
   AG4.SP3 := FALSE;
   AG4.SP4 := FALSE;
   AG4.FC6_STATUS := W#16#0;
   AG4.FC6_DPSTATUS := B#16#0;
   AG4.FC5_STATUS := W#16#0;
   AG4.SP5 := W#16#0;
   AG4.SFC20_1_RET_VAL := 0;
   AG4.SFC20_2_RET_VAL := 0;
   AG4.SFC20_3_RET_VAL := 0;
   AG4.SFC20_4_RET_VAL := 0;
   AG4.SFC20_5_RET_VAL := 0;
   AG4.SFC20_6_RET_VAL := 0;
   AG4.SFC20_7_RET_VAL := 0;
   AG4.SFC20_8_RET_VAL := 0;
   AG4.SFC20_9_RET_VAL := 0;
   AG4.SFC20_10_RET_VAL := 0;
   AG4.SP[0] := W#16#0;
   AG4.SP[1] := W#16#0;
   AG4.SP[2] := W#16#0;
   AG4.SP[3] := W#16#0;
   AG4.SP[4] := W#16#0;
   AG4.SP[5] := W#16#0;
   AG4.SP[6] := W#16#0;
   AG4.SP[7] := W#16#0;
   AG4.SP[8] := W#16#0;
   AG4.SP[9] := W#16#0;
   AG5.FC6_NDR := FALSE;
   AG5.FC6_ERROR := FALSE;
   AG5.SP1 := FALSE;
   AG5.SP2 := FALSE;
   AG5.FC5_NDR := FALSE;
   AG5.FC5_ERROR := FALSE;
   AG5.SP3 := FALSE;
   AG5.SP4 := FALSE;
   AG5.FC6_STATUS := W#16#0;
   AG5.FC6_DPSTATUS := B#16#0;
   AG5.FC5_STATUS := W#16#0;
   AG5.SP5 := W#16#0;
   AG5.SFC20_1_RET_VAL := 0;
   AG5.SFC20_2_RET_VAL := 0;
   AG5.SFC20_3_RET_VAL := 0;
   AG5.SFC20_4_RET_VAL := 0;
   AG5.SFC20_5_RET_VAL := 0;
   AG5.SFC20_6_RET_VAL := 0;
   AG5.SFC20_7_RET_VAL := 0;
   AG5.SFC20_8_RET_VAL := 0;
   AG5.SFC20_9_RET_VAL := 0;
   AG5.SFC20_10_RET_VAL := 0;
   AG5.SP[0] := W#16#0;
   AG5.SP[1] := W#16#0;
   AG5.SP[2] := W#16#0;
   AG5.SP[3] := W#16#0;
   AG5.SP[4] := W#16#0;
   AG5.SP[5] := W#16#0;
   AG5.SP[6] := W#16#0;
   AG5.SP[7] := W#16#0;
   AG5.SP[8] := W#16#0;
   AG5.SP[9] := W#16#0;
   AG6.FC6_NDR := FALSE;
   AG6.FC6_ERROR := FALSE;
   AG6.SP1 := FALSE;
   AG6.SP2 := FALSE;
   AG6.FC5_NDR := FALSE;
   AG6.FC5_ERROR := FALSE;
   AG6.SP3 := FALSE;
   AG6.SP4 := FALSE;
   AG6.FC6_STATUS := W#16#0;
   AG6.FC6_DPSTATUS := B#16#0;
   AG6.FC5_STATUS := W#16#0;
   AG6.SP5 := W#16#0;
   AG6.SFC20_1_RET_VAL := 0;
   AG6.SFC20_2_RET_VAL := 0;
   AG6.SFC20_3_RET_VAL := 0;
   AG6.SFC20_4_RET_VAL := 0;
   AG6.SFC20_5_RET_VAL := 0;
   AG6.SFC20_6_RET_VAL := 0;
   AG6.SFC20_7_RET_VAL := 0;
   AG6.SFC20_8_RET_VAL := 0;
   AG6.SFC20_9_RET_VAL := 0;
   AG6.SFC20_10_RET_VAL := 0;
   AG6.SP[0] := W#16#0;
   AG6.SP[1] := W#16#0;
   AG6.SP[2] := W#16#0;
   AG6.SP[3] := W#16#0;
   AG6.SP[4] := W#16#0;
   AG6.SP[5] := W#16#0;
   AG6.SP[6] := W#16#0;
   AG6.SP[7] := W#16#0;
   AG6.SP[8] := W#16#0;
   AG6.SP[9] := W#16#0;
   AG7.FC6_NDR := FALSE;
   AG7.FC6_ERROR := FALSE;
   AG7.SP1 := FALSE;
   AG7.SP2 := FALSE;
   AG7.FC5_NDR := FALSE;
   AG7.FC5_ERROR := FALSE;
   AG7.SP3 := FALSE;
   AG7.SP4 := FALSE;
   AG7.FC6_STATUS := W#16#0;
   AG7.FC6_DPSTATUS := B#16#0;
   AG7.FC5_STATUS := W#16#0;
   AG7.SP5 := W#16#0;
   AG7.SFC20_1_RET_VAL := 0;
   AG7.SFC20_2_RET_VAL := 0;
   AG7.SFC20_3_RET_VAL := 0;
   AG7.SFC20_4_RET_VAL := 0;
   AG7.SFC20_5_RET_VAL := 0;
   AG7.SFC20_6_RET_VAL := 0;
   AG7.SFC20_7_RET_VAL := 0;
   AG7.SFC20_8_RET_VAL := 0;
   AG7.SFC20_9_RET_VAL := 0;
   AG7.SFC20_10_RET_VAL := 0;
   AG7.SP[0] := W#16#0;
   AG7.SP[1] := W#16#0;
   AG7.SP[2] := W#16#0;
   AG7.SP[3] := W#16#0;
   AG7.SP[4] := W#16#0;
   AG7.SP[5] := W#16#0;
   AG7.SP[6] := W#16#0;
   AG7.SP[7] := W#16#0;
   AG7.SP[8] := W#16#0;
   AG7.SP[9] := W#16#0;
   SP[0] := W#16#0;
   SP[1] := W#16#0;
   SP[2] := W#16#0;
   SP[3] := W#16#0;
   SP[4] := W#16#0;
   SP[5] := W#16#0;
   SP[6] := W#16#0;
   SP[7] := W#16#0;
   SP[8] := W#16#0;
   SP[9] := W#16#0;
   SP[10] := W#16#0;
   SP[11] := W#16#0;
   SP[12] := W#16#0;
   SP[13] := W#16#0;
   SP[14] := W#16#0;
   SP[15] := W#16#0;
   SP[16] := W#16#0;
   SP[17] := W#16#0;
   SP[18] := W#16#0;
   SP[19] := W#16#0;
   SP[20] := W#16#0;
   SP[21] := W#16#0;
   SP[22] := W#16#0;
   SP[23] := W#16#0;
   SP[24] := W#16#0;
   SP[25] := W#16#0;
   SP[26] := W#16#0;
   SP[27] := W#16#0;
   SP[28] := W#16#0;
   SP[29] := W#16#0;
   SP[30] := W#16#0;
   SP[31] := W#16#0;
   SP[32] := W#16#0;
   SP[33] := W#16#0;
   SP[34] := W#16#0;
   SP[35] := W#16#0;
   SP[36] := W#16#0;
   SP[37] := W#16#0;
   SP[38] := W#16#0;
   SP[39] := W#16#0;
   SP[40] := W#16#0;
   SP[41] := W#16#0;
   SP[42] := W#16#0;
   SP[43] := W#16#0;
   SP[44] := W#16#0;
   SP[45] := W#16#0;
   SP[46] := W#16#0;
   SP[47] := W#16#0;
   SP[48] := W#16#0;
   SP[49] := W#16#0;
   SP[50] := W#16#0;
   SP[51] := W#16#0;
   SP[52] := W#16#0;
   SP[53] := W#16#0;
   SP[54] := W#16#0;
   SP[55] := W#16#0;
   SP[56] := W#16#0;
   SP[57] := W#16#0;
   SP[58] := W#16#0;
   SP[59] := W#16#0;
   SP[60] := W#16#0;
   SP[61] := W#16#0;
   SP[62] := W#16#0;
   SP[63] := W#16#0;
   SP[64] := W#16#0;
   SP[65] := W#16#0;
   SP[66] := W#16#0;
   SP[67] := W#16#0;
   SP[68] := W#16#0;
   SP[69] := W#16#0;
   SP[70] := W#16#0;
   SP[71] := W#16#0;
   SP[72] := W#16#0;
   SP[73] := W#16#0;
   SP[74] := W#16#0;
   CTYPE_RET_VAL[0] := 0;
   CTYPE_RET_VAL[1] := 0;
   CTYPE_RET_VAL[2] := 0;
   CTYPE_RET_VAL[3] := 0;
   CTYPE_RET_VAL[4] := 0;
   CTYPE_RET_VAL[5] := 0;
   CTYPE_RET_VAL[6] := 0;
   CTYPE_RET_VAL[7] := 0;
   CTYPE_RET_VAL[8] := 0;
   CTYPE_RET_VAL[9] := 0;
   CTYPE_RET_VAL[10] := 0;
   CTYPE_RET_VAL[11] := 0;
   CTYPE_RET_VAL[12] := 0;
   CTYPE_RET_VAL[13] := 0;
   CTYPE_RET_VAL[14] := 0;
   CTYPE_RET_VAL[15] := 0;
   CTYPE_RET_VAL[16] := 0;
   CTYPE_RET_VAL[17] := 0;
   CTYPE_RET_VAL[18] := 0;
   CTYPE_RET_VAL[19] := 0;
   CTYPE_RET_VAL[20] := 0;
   CTYPE_RET_VAL[21] := 0;
   CTYPE_RET_VAL[22] := 0;
   CTYPE_RET_VAL[23] := 0;
   CTYPE_RET_VAL[24] := 0;
   CTYPE_RET_VAL[25] := 0;
   CTYPE_RET_VAL[26] := 0;
   CTYPE_RET_VAL[27] := 0;
   CTYPE_RET_VAL[28] := 0;
   CTYPE_RET_VAL[29] := 0;
   CTYPE_RET_VAL[30] := 0;
   CTYPE_RET_VAL[31] := 0;
   CTYPE_RET_VAL[32] := 0;
   CTYPE_RET_VAL[33] := 0;
   CTYPE_RET_VAL[34] := 0;
   CTYPE_RET_VAL[35] := 0;
   CTYPE_RET_VAL[36] := 0;
   CTYPE_RET_VAL[37] := 0;
   CTYPE_RET_VAL[38] := 0;
   CTYPE_RET_VAL[39] := 0;
   CTYPE_RET_VAL[40] := 0;
   CTYPE_RET_VAL[41] := 0;
   CTYPE_RET_VAL[42] := 0;
   CTYPE_RET_VAL[43] := 0;
   CTYPE_RET_VAL[44] := 0;
   CTYPE_RET_VAL[45] := 0;
   CTYPE_RET_VAL[46] := 0;
   CTYPE_RET_VAL[47] := 0;
   CTYPE_RET_VAL[48] := 0;
   CTYPE_RET_VAL[49] := 0;
   CTYPE_RET_VAL[50] := 0;
   CTYPE_RET_VAL[51] := 0;
   CTYPE_RET_VAL[52] := 0;
   CTYPE_RET_VAL[53] := 0;
   CTYPE_RET_VAL[54] := 0;
   CTYPE_RET_VAL[55] := 0;
   CTYPE_RET_VAL[56] := 0;
   CTYPE_RET_VAL[57] := 0;
   CTYPE_RET_VAL[58] := 0;
   CTYPE_RET_VAL[59] := 0;
   CTYPE_RET_VAL[60] := 0;
   CTYPE_RET_VAL[61] := 0;
   CTYPE_RET_VAL[62] := 0;
   CTYPE_RET_VAL[63] := 0;
   CTYPE_RET_VAL[64] := 0;
   CTYPE_RET_VAL[65] := 0;
   CTYPE_RET_VAL[66] := 0;
   CTYPE_RET_VAL[67] := 0;
   CTYPE_RET_VAL[68] := 0;
   CTYPE_RET_VAL[69] := 0;
   CTYPE_RET_VAL[70] := 0;
   CTYPE_RET_VAL[71] := 0;
   CTYPE_RET_VAL[72] := 0;
   CTYPE_RET_VAL[73] := 0;
   CTYPE_RET_VAL[74] := 0;
   CTYPE_RET_VAL[75] := 0;
   CTYPE_RET_VAL[76] := 0;
   CTYPE_RET_VAL[77] := 0;
   CTYPE_RET_VAL[78] := 0;
   CTYPE_RET_VAL[79] := 0;
   CTYPE_RET_VAL[80] := 0;
   CTYPE_RET_VAL[81] := 0;
   CTYPE_RET_VAL[82] := 0;
   CTYPE_RET_VAL[83] := 0;
   CTYPE_RET_VAL[84] := 0;
   CTYPE_RET_VAL[85] := 0;
   CTYPE_RET_VAL[86] := 0;
   CTYPE_RET_VAL[87] := 0;
   CTYPE_RET_VAL[88] := 0;
   CTYPE_RET_VAL[89] := 0;
   CTYPE_RET_VAL[90] := 0;
   CTYPE_RET_VAL[91] := 0;
   CTYPE_RET_VAL[92] := 0;
   CTYPE_RET_VAL[93] := 0;
   CTYPE_RET_VAL[94] := 0;
   CTYPE_RET_VAL[95] := 0;
   CTYPE_RET_VAL[96] := 0;
   CTYPE_RET_VAL[97] := 0;
   CTYPE_RET_VAL[98] := 0;
   CTYPE_RET_VAL[99] := 0;
   MES_RET_VAL1[0] := 0;
   MES_RET_VAL1[1] := 0;
   MES_RET_VAL1[2] := 0;
   MES_RET_VAL1[3] := 0;
   MES_RET_VAL1[4] := 0;
   MES_RET_VAL1[5] := 0;
   MES_RET_VAL1[6] := 0;
   MES_RET_VAL1[7] := 0;
   MES_RET_VAL1[8] := 0;
   MES_RET_VAL1[9] := 0;
   MES_RET_VAL1[10] := 0;
   MES_RET_VAL1[11] := 0;
   MES_RET_VAL1[12] := 0;
   MES_RET_VAL1[13] := 0;
   MES_RET_VAL1[14] := 0;
   MES_RET_VAL1[15] := 0;
   MES_RET_VAL1[16] := 0;
   MES_RET_VAL1[17] := 0;
   MES_RET_VAL1[18] := 0;
   MES_RET_VAL1[19] := 0;
   MES_RET_VAL1[20] := 0;
   MES_RET_VAL1[21] := 0;
   MES_RET_VAL1[22] := 0;
   MES_RET_VAL1[23] := 0;
   MES_RET_VAL1[24] := 0;
   MES_RET_VAL1[25] := 0;
   MES_RET_VAL1[26] := 0;
   MES_RET_VAL1[27] := 0;
   MES_RET_VAL1[28] := 0;
   MES_RET_VAL1[29] := 0;
   MES_RET_VAL1[30] := 0;
   MES_RET_VAL1[31] := 0;
   MES_RET_VAL1[32] := 0;
   MES_RET_VAL1[33] := 0;
   MES_RET_VAL1[34] := 0;
   MES_RET_VAL1[35] := 0;
   MES_RET_VAL1[36] := 0;
   MES_RET_VAL1[37] := 0;
   MES_RET_VAL1[38] := 0;
   MES_RET_VAL1[39] := 0;
   MES_RET_VAL1[40] := 0;
   MES_RET_VAL1[41] := 0;
   MES_RET_VAL1[42] := 0;
   MES_RET_VAL1[43] := 0;
   MES_RET_VAL1[44] := 0;
   MES_RET_VAL1[45] := 0;
   MES_RET_VAL1[46] := 0;
   MES_RET_VAL1[47] := 0;
   MES_RET_VAL1[48] := 0;
   MES_RET_VAL1[49] := 0;
   MES_RET_VAL1[50] := 0;
   MES_RET_VAL1[51] := 0;
   MES_RET_VAL1[52] := 0;
   MES_RET_VAL1[53] := 0;
   MES_RET_VAL1[54] := 0;
   MES_RET_VAL1[55] := 0;
   MES_RET_VAL1[56] := 0;
   MES_RET_VAL1[57] := 0;
   MES_RET_VAL1[58] := 0;
   MES_RET_VAL1[59] := 0;
   MES_RET_VAL1[60] := 0;
   MES_RET_VAL1[61] := 0;
   MES_RET_VAL1[62] := 0;
   MES_RET_VAL1[63] := 0;
   MES_RET_VAL1[64] := 0;
   MES_RET_VAL1[65] := 0;
   MES_RET_VAL1[66] := 0;
   MES_RET_VAL1[67] := 0;
   MES_RET_VAL1[68] := 0;
   MES_RET_VAL1[69] := 0;
   MES_RET_VAL1[70] := 0;
   MES_RET_VAL1[71] := 0;
   MES_RET_VAL1[72] := 0;
   MES_RET_VAL1[73] := 0;
   MES_RET_VAL1[74] := 0;
   MES_RET_VAL1[75] := 0;
   MES_RET_VAL1[76] := 0;
   MES_RET_VAL1[77] := 0;
   MES_RET_VAL1[78] := 0;
   MES_RET_VAL1[79] := 0;
   MES_RET_VAL1[80] := 0;
   MES_RET_VAL1[81] := 0;
   MES_RET_VAL1[82] := 0;
   MES_RET_VAL1[83] := 0;
   MES_RET_VAL1[84] := 0;
   MES_RET_VAL1[85] := 0;
   MES_RET_VAL1[86] := 0;
   MES_RET_VAL1[87] := 0;
   MES_RET_VAL1[88] := 0;
   MES_RET_VAL1[89] := 0;
   MES_RET_VAL1[90] := 0;
   MES_RET_VAL1[91] := 0;
   MES_RET_VAL1[92] := 0;
   MES_RET_VAL1[93] := 0;
   MES_RET_VAL1[94] := 0;
   MES_RET_VAL1[95] := 0;
   MES_RET_VAL1[96] := 0;
   MES_RET_VAL1[97] := 0;
   MES_RET_VAL1[98] := 0;
   MES_RET_VAL1[99] := 0;
   MES_RET_VAL1[100] := 0;
   MES_RET_VAL1[101] := 0;
   MES_RET_VAL1[102] := 0;
   MES_RET_VAL1[103] := 0;
   MES_RET_VAL1[104] := 0;
   MES_RET_VAL1[105] := 0;
   MES_RET_VAL1[106] := 0;
   MES_RET_VAL1[107] := 0;
   MES_RET_VAL1[108] := 0;
   MES_RET_VAL1[109] := 0;
   MES_RET_VAL1[110] := 0;
   MES_RET_VAL1[111] := 0;
   MES_RET_VAL1[112] := 0;
   MES_RET_VAL1[113] := 0;
   MES_RET_VAL1[114] := 0;
   MES_RET_VAL1[115] := 0;
   MES_RET_VAL1[116] := 0;
   MES_RET_VAL1[117] := 0;
   MES_RET_VAL1[118] := 0;
   MES_RET_VAL1[119] := 0;
   MES_RET_VAL1[120] := 0;
   MES_RET_VAL1[121] := 0;
   MES_RET_VAL1[122] := 0;
   MES_RET_VAL1[123] := 0;
   MES_RET_VAL1[124] := 0;
   MES_RET_VAL1[125] := 0;
   MES_RET_VAL1[126] := 0;
   MES_RET_VAL1[127] := 0;
   MES_RET_VAL1[128] := 0;
   MES_RET_VAL1[129] := 0;
   MES_RET_VAL1[130] := 0;
   MES_RET_VAL1[131] := 0;
   MES_RET_VAL1[132] := 0;
   MES_RET_VAL1[133] := 0;
   MES_RET_VAL1[134] := 0;
   MES_RET_VAL1[135] := 0;
   MES_RET_VAL1[136] := 0;
   MES_RET_VAL1[137] := 0;
   MES_RET_VAL1[138] := 0;
   MES_RET_VAL1[139] := 0;
   MES_RET_VAL1[140] := 0;
   MES_RET_VAL1[141] := 0;
   MES_RET_VAL1[142] := 0;
   MES_RET_VAL1[143] := 0;
   MES_RET_VAL1[144] := 0;
   MES_RET_VAL1[145] := 0;
   MES_RET_VAL1[146] := 0;
   MES_RET_VAL1[147] := 0;
   MES_RET_VAL1[148] := 0;
   MES_RET_VAL1[149] := 0;
   MES_RET_VAL1[150] := 0;
   MES_RET_VAL1[151] := 0;
   MES_RET_VAL1[152] := 0;
   MES_RET_VAL1[153] := 0;
   MES_RET_VAL1[154] := 0;
   MES_RET_VAL1[155] := 0;
   MES_RET_VAL1[156] := 0;
   MES_RET_VAL1[157] := 0;
   MES_RET_VAL1[158] := 0;
   MES_RET_VAL1[159] := 0;
   MES_RET_VAL1[160] := 0;
   MES_RET_VAL1[161] := 0;
   MES_RET_VAL1[162] := 0;
   MES_RET_VAL1[163] := 0;
   MES_RET_VAL1[164] := 0;
   MES_RET_VAL1[165] := 0;
   MES_RET_VAL1[166] := 0;
   MES_RET_VAL1[167] := 0;
   MES_RET_VAL1[168] := 0;
   MES_RET_VAL1[169] := 0;
   MES_RET_VAL1[170] := 0;
   MES_RET_VAL1[171] := 0;
   MES_RET_VAL1[172] := 0;
   MES_RET_VAL1[173] := 0;
   MES_RET_VAL1[174] := 0;
   MES_RET_VAL1[175] := 0;
   MES_RET_VAL1[176] := 0;
   MES_RET_VAL1[177] := 0;
   MES_RET_VAL1[178] := 0;
   MES_RET_VAL1[179] := 0;
   MES_RET_VAL1[180] := 0;
   MES_RET_VAL1[181] := 0;
   MES_RET_VAL1[182] := 0;
   MES_RET_VAL1[183] := 0;
   MES_RET_VAL1[184] := 0;
   MES_RET_VAL1[185] := 0;
   MES_RET_VAL1[186] := 0;
   MES_RET_VAL1[187] := 0;
   MES_RET_VAL1[188] := 0;
   MES_RET_VAL1[189] := 0;
   MES_RET_VAL1[190] := 0;
   MES_RET_VAL1[191] := 0;
   MES_RET_VAL1[192] := 0;
   MES_RET_VAL1[193] := 0;
   MES_RET_VAL1[194] := 0;
   MES_RET_VAL1[195] := 0;
   MES_RET_VAL1[196] := 0;
   MES_RET_VAL1[197] := 0;
   MES_RET_VAL1[198] := 0;
   MES_RET_VAL1[199] := 0;
END_DATA_BLOCK

DATA_BLOCK DB 59
TITLE =
VERSION : 0.1


